LIN {X 0,Y 395.953,Z 958.615,A -85,B 0,C 180,E1 18668.249,E2 18668.249} C_VEL
LIN {X 0,Y 392.265,Z 977.783,A -85,B 0,C 180,E1 18665.892,E2 18665.892} C_VEL
LIN {X 0,Y 388.745,Z 995.88,A -85,B 0,C 180,E1 18663.291,E2 18663.291} C_VEL
LIN {X 0,Y 385.497,Z 1013.366,A -85,B 0,C 180,E1 18660.383,E2 18660.383} C_VEL
LIN {X 0,Y 382.925,Z 1028.309,A -85,B 0,C 180,E1 18657.527,E2 18657.527} C_VEL
LIN {X 0,Y 380.669,Z 1042.529,A -85,B 0,C 180,E1 18654.354,E2 18654.354} C_VEL
LIN {X 0,Y 378.971,Z 1054.652,A -85,B 0,C 180,E1 18651.19,E2 18651.19} C_VEL
LIN {X 0,Y 377.875,Z 1063.785,A -85,B 0,C 180,E1 18648.353,E2 18648.353} C_VEL
LIN {X 0,Y 376.991,Z 1072.565,A -85,B 0,C 180,E1 18645.065,E2 18645.065} C_VEL
LIN {X 0,Y 376.551,Z 1078.821,A -85,B 0,C 180,E1 18642.109,E2 18642.109} C_VEL
LIN {X 0,Y 376.293,Z 1084.179,A -85,B 0,C 180,E1 18638.865,E2 18638.865} C_VEL
LIN {X 0,Y 376.216,Z 1087.581,A -85,B 0,C 180,E1 18635.796,E2 18635.796} C_VEL
LIN {X 0,Y 376.187,Z 1089.458,A -85,B 0,C 180,E1 18633.047,E2 18633.047} C_VEL
LIN {X 0,Y 376.206,Z 1090.251,A -85,B 0,C 180,E1 18630,E2 18630} C_VEL
LIN {X 0,Y 376.187,Z 1089.461,A -85,B 0,C 180,E1 18626.953,E2 18626.953} C_VEL
LIN {X 0,Y 376.215,Z 1087.586,A -85,B 0,C 180,E1 18624.204,E2 18624.204} C_VEL
LIN {X 0,Y 376.297,Z 1083.964,A -85,B 0,C 180,E1 18620.98,E2 18620.98} C_VEL
LIN {X 0,Y 376.573,Z 1078.539,A -85,B 0,C 180,E1 18617.736,E2 18617.736} C_VEL
LIN {X 0,Y 377.088,Z 1071.485,A -85,B 0,C 180,E1 18614.466,E2 18614.466} C_VEL
LIN {X 0,Y 378,Z 1062.621,A -85,B 0,C 180,E1 18611.253,E2 18611.253} C_VEL
LIN {X 0,Y 379.354,Z 1051.878,A -85,B 0,C 180,E1 18608.021,E2 18608.021} C_VEL
LIN {X 0,Y 380.971,Z 1040.525,A -85,B 0,C 180,E1 18605.17,E2 18605.17} C_VEL
LIN {X 0,Y 383.492,Z 1024.877,A -85,B 0,C 180,E1 18601.792,E2 18601.792} C_VEL
LIN {X 0,Y 386.339,Z 1008.954,A -85,B 0,C 180,E1 18598.828,E2 18598.828} C_VEL
LIN {X 0,Y 389.531,Z 991.792,A -85,B 0,C 180,E1 18596.091,E2 18596.091} C_VEL
LIN {X 0,Y 393.28,Z 972.35,A -85,B 0,C 180,E1 18593.412,E2 18593.412} C_VEL
LIN {X 0,Y 397.008,Z 953.443,A -85,B 0,C 180,E1 18591.163,E2 18591.163} C_VEL
LIN {X 0,Y 400.919,Z 932.814,A -85,B 0,C 180,E1 18589.082,E2 18589.082} C_VEL
LIN {X 0,Y 404.892,Z 911.134,A -85,B 0,C 180,E1 18587.226,E2 18587.226} C_VEL
LIN {X 0,Y 408.617,Z 889.656,A -85,B 0,C 180,E1 18585.685,E2 18585.685} C_VEL
LIN {X 0,Y 411.957,Z 868.031,A -85,B 0,C 180,E1 18584.424,E2 18584.424} C_VEL
LIN {X 0,Y 415.071,Z 845.276,A -85,B 0,C 180,E1 18583.348,E2 18583.348} C_VEL
LIN {X 0,Y 417.607,Z 823.088,A -85,B 0,C 180,E1 18582.55,E2 18582.55} C_VEL
LIN {X 0,Y 419.585,Z 798.577,A -85,B 0,C 180,E1 18581.9,E2 18581.9} C_VEL
LIN {X 0,Y 428.412,Z 598.085,A -85,B 0,C 180,E1 18577.889,E2 18577.889} C_VEL
LIN {X 0,Y 432.313,Z 505.731,A -85,B 0,C 180,E1 18576.053,E2 18576.053} C_VEL
LIN {X 0,Y 430.788,Z 488.115,A -85,B 0,C 180,E1 18575.366,E2 18575.366} C_VEL
LIN {X 0,Y 419.802,Z 470.98,A -85,B 0,C 180,E1 18573.134,E2 18573.134} C_VEL
LIN {X 0,Y 416.485,Z 465.848,A -85,B 0,C 180,E1 18572.368,E2 18572.368} C_VEL
LIN {X 0,Y 408.57,Z 450.774,A -85,B 0,C 180,E1 18569.303,E2 18569.303} C_VEL
LIN {X 0,Y 402.669,Z 440.538,A -85,B 0,C 180,E1 18566.866,E2 18566.866} C_VEL
LIN {X 0,Y 398.101,Z 432.532,A -85,B 0,C 180,E1 18564.798,E2 18564.798} C_VEL
LIN {X 0,Y 394.857,Z 427.301,A -85,B 0,C 180,E1 18563.267,E2 18563.267} C_VEL
LIN {X 0,Y 391.803,Z 422.309,A -85,B 0,C 180,E1 18561.717,E2 18561.717} C_VEL
LIN {X 0,Y 389.222,Z 418.314,A -85,B 0,C 180,E1 18560.34,E2 18560.34} C_VEL
LIN {X 0,Y 388.405,Z 416.892,A -85,B 0,C 180,E1 18559.864,E2 18559.864} C_VEL
LIN {X 0,Y 385.879,Z 413.274,A -85,B 0,C 180,E1 18558.428,E2 18558.428} C_VEL
LIN {X 0,Y 385.059,Z 411.546,A -85,B 0,C 180,E1 18557.842,E2 18557.842} C_VEL
LIN {X 0,Y 382.366,Z 408.271,A -85,B 0,C 180,E1 18556.248,E2 18556.248} C_VEL
LIN {X 0,Y 381.062,Z 405.625,A -85,B 0,C 180,E1 18555.211,E2 18555.211} C_VEL
LIN {X 0,Y 378.291,Z 402.297,A -85,B 0,C 180,E1 18553.294,E2 18553.294} C_VEL
LIN {X 0,Y 377.687,Z 400.258,A -85,B 0,C 180,E1 18552.347,E2 18552.347} C_VEL
LIN {X 0,Y 377.63,Z 399.995,A -85,B 0,C 180,E1 18548.987,E2 18548.987} C_VEL
LIN {X 0,Y 377.616,Z 399.995,A -85,B 0,C 180,E1 18545.165,E2 18545.165} C_VEL
LIN {X 0,Y 377.616,Z 399.993,A -85,B 0,C 180,E1 18541.062,E2 18541.062} C_VEL
LIN {X 0,Y 377.616,Z 399.992,A -85,B 0,C 180,E1 18536.964,E2 18536.964} C_VEL
LIN {X 0,Y 377.616,Z 399.989,A -85,B 0,C 180,E1 18532.851,E2 18532.851} C_VEL
LIN {X 0,Y 377.623,Z 399.989,A -85,B 0,C 180,E1 18528.855,E2 18528.855} C_VEL
LIN {X 0,Y 377.637,Z 399.988,A -85,B 0,C 180,E1 18524.961,E2 18524.961} C_VEL
LIN {X 0,Y 377.652,Z 399.988,A -85,B 0,C 180,E1 18520.995,E2 18520.995} C_VEL
LIN {X 0,Y 377.652,Z 400.221,A -85,B 0,C 180,E1 18518.08,E2 18518.08} C_VEL
LIN {X 0,Y 379.501,Z 404.243,A -85,B 0,C 180,E1 18516.062,E2 18516.062} C_VEL
LIN {X 0,Y 381.324,Z 406.087,A -85,B 0,C 180,E1 18514.863,E2 18514.863} C_VEL
LIN {X 0,Y 382.924,Z 409.558,A -85,B 0,C 180,E1 18513.48,E2 18513.48} C_VEL
LIN {X 0,Y 384.703,Z 411.566,A -85,B 0,C 180,E1 18512.409,E2 18512.409} C_VEL
LIN {X 0,Y 386.855,Z 415.598,A -85,B 0,C 180,E1 18510.879,E2 18510.879} C_VEL
LIN {X 0,Y 388.007,Z 417.315,A -85,B 0,C 180,E1 18510.175,E2 18510.175} C_VEL
LIN {X 0,Y 391.15,Z 422.892,A -85,B 0,C 180,E1 18508.225,E2 18508.225} C_VEL
LIN {X 0,Y 393.971,Z 427.927,A -85,B 0,C 180,E1 18506.583,E2 18506.583} C_VEL
LIN {X 0,Y 396.924,Z 433.413,A -85,B 0,C 180,E1 18504.946,E2 18504.946} C_VEL
LIN {X 0,Y 401.486,Z 441.984,A -85,B 0,C 180,E1 18502.579,E2 18502.579} C_VEL
LIN {X 0,Y 407.169,Z 453.602,A -85,B 0,C 180,E1 18499.771,E2 18499.771} C_VEL
LIN {X 0,Y 413.175,Z 466.753,A -85,B 0,C 180,E1 18496.956,E2 18496.956} C_VEL
LIN {X 0,Y 414.811,Z 470.097,A -85,B 0,C 180,E1 18496.371,E2 18496.371} C_VEL
LIN {X 0,Y 422.176,Z 481.769,A -85,B 0,C 180,E1 18494.82,E2 18494.82} C_VEL
LIN {X 0,Y 426.207,Z 512.164,A -85,B 0,C 180,E1 18493.447,E2 18493.447} C_VEL
LIN {X 0,Y 419.079,Z 748.452,A -85,B 0,C 180,E1 18489.374,E2 18489.374} C_VEL
LIN {X 0,Y 417.798,Z 768.888,A -85,B 0,C 180,E1 18488.782,E2 18488.782} C_VEL
LIN {X 0,Y 415.904,Z 788.515,A -85,B 0,C 180,E1 18487.984,E2 18487.984} C_VEL
LIN {X 0,Y 413.573,Z 806.905,A -85,B 0,C 180,E1 18487.013,E2 18487.013} C_VEL
LIN {X 0,Y 410.543,Z 825.493,A -85,B 0,C 180,E1 18485.769,E2 18485.769} C_VEL
LIN {X 0,Y 407.124,Z 843.157,A -85,B 0,C 180,E1 18484.308,E2 18484.308} C_VEL
LIN {X 0,Y 403.192,Z 860.843,A -85,B 0,C 180,E1 18482.525,E2 18482.525} C_VEL
LIN {X 0,Y 399.371,Z 876.448,A -85,B 0,C 180,E1 18480.622,E2 18480.622} C_VEL
LIN {X 0,Y 395.306,Z 891.616,A -85,B 0,C 180,E1 18478.393,E2 18478.393} C_VEL
LIN {X 0,Y 393.493,Z 897.983,A -85,B 0,C 180,E1 18477.31,E2 18477.31} C_VEL
LIN {X 0,Y 391.285,Z 902.98,A -85,B 0,C 180,E1 18476.504,E2 18476.504} C_VEL
LIN {X 0,Y 382.56,Z 915.406,A -85,B 0,C 180,E1 18474.535,E2 18474.535} C_VEL
LIN {X 0,Y 380.407,Z 919.642,A -85,B 0,C 180,E1 18473.623,E2 18473.623} C_VEL
LIN {X 0,Y 377.243,Z 930.013,A -85,B 0,C 180,E1 18470.803,E2 18470.803} C_VEL
LIN {X 0,Y 374.496,Z 939.227,A -85,B 0,C 180,E1 18467.72,E2 18467.72} C_VEL
LIN {X 0,Y 372.489,Z 946.593,A -85,B 0,C 180,E1 18464.615,E2 18464.615} C_VEL
LIN {X 0,Y 370.947,Z 952.787,A -85,B 0,C 180,E1 18461.191,E2 18461.191} C_VEL
LIN {X 0,Y 370.038,Z 957.128,A -85,B 0,C 180,E1 18457.765,E2 18457.765} C_VEL
LIN {X 0,Y 369.539,Z 959.825,A -85,B 0,C 180,E1 18454.345,E2 18454.345} C_VEL
LIN {X 0,Y 369.359,Z 960.993,A -85,B 0,C 180,E1 18450.931,E2 18450.931} C_VEL
LIN {X 0,Y 369.406,Z 960.688,A -85,B 0,C 180,E1 18447.518,E2 18447.518} C_VEL
LIN {X 0,Y 369.689,Z 959.027,A -85,B 0,C 180,E1 18444.257,E2 18444.257} C_VEL
LIN {X 0,Y 370.331,Z 955.662,A -85,B 0,C 180,E1 18440.834,E2 18440.834} C_VEL
LIN {X 0,Y 371.377,Z 950.872,A -85,B 0,C 180,E1 18437.562,E2 18437.562} C_VEL
LIN {X 0,Y 373.071,Z 944.401,A -85,B 0,C 180,E1 18434.295,E2 18434.295} C_VEL
LIN {X 0,Y 375.304,Z 936.512,A -85,B 0,C 180,E1 18431.194,E2 18431.194} C_VEL
LIN {X 0,Y 378.123,Z 927.246,A -85,B 0,C 180,E1 18428.272,E2 18428.272} C_VEL
LIN {X 0,Y 381.56,Z 916,A -85,B 0,C 180,E1 18425.409,E2 18425.409} C_VEL
LIN {X 0,Y 385.313,Z 903.641,A -85,B 0,C 180,E1 18422.825,E2 18422.825} C_VEL
LIN {X 0,Y 389.315,Z 890.006,A -85,B 0,C 180,E1 18420.455,E2 18420.455} C_VEL
LIN {X 0,Y 393.299,Z 875.817,A -85,B 0,C 180,E1 18418.392,E2 18418.392} C_VEL
LIN {X 0,Y 397.328,Z 859.912,A -85,B 0,C 180,E1 18416.471,E2 18416.471} C_VEL
LIN {X 0,Y 401.185,Z 843.001,A -85,B 0,C 180,E1 18414.784,E2 18414.784} C_VEL
LIN {X 0,Y 404.796,Z 824.782,A -85,B 0,C 180,E1 18413.291,E2 18413.291} C_VEL
LIN {X 0,Y 407.854,Z 806.475,A -85,B 0,C 180,E1 18412.073,E2 18412.073} C_VEL
LIN {X 0,Y 410.397,Z 786.949,A -85,B 0,C 180,E1 18411.055,E2 18411.055} C_VEL
LIN {X 0,Y 412.29,Z 767.123,A -85,B 0,C 180,E1 18410.278,E2 18410.278} C_VEL
LIN {X 0,Y 413.536,Z 745.732,A -85,B 0,C 180,E1 18409.69,E2 18409.69} C_VEL
LIN {X 0,Y 420.978,Z 512.412,A -85,B 0,C 180,E1 18405.623,E2 18405.623} C_VEL
LIN {X 0,Y 417.279,Z 485.839,A -85,B 0,C 180,E1 18404.353,E2 18404.353} C_VEL
LIN {X 0,Y 406.186,Z 468.485,A -85,B 0,C 180,E1 18401.843,E2 18401.843} C_VEL
LIN {X 0,Y 399.907,Z 454.656,A -85,B 0,C 180,E1 18398.732,E2 18398.732} C_VEL
LIN {X 0,Y 393.543,Z 441.944,A -85,B 0,C 180,E1 18395.4,E2 18395.4} C_VEL
LIN {X 0,Y 388.521,Z 432.569,A -85,B 0,C 180,E1 18392.539,E2 18392.539} C_VEL
LIN {X 0,Y 385.533,Z 427.329,A -85,B 0,C 180,E1 18390.725,E2 18390.725} C_VEL
LIN {X 0,Y 382.719,Z 422.434,A -85,B 0,C 180,E1 18388.903,E2 18388.903} C_VEL
LIN {X 0,Y 380.492,Z 418.59,A -85,B 0,C 180,E1 18387.351,E2 18387.351} C_VEL
LIN {X 0,Y 379.383,Z 417.056,A -85,B 0,C 180,E1 18386.618,E2 18386.618} C_VEL
LIN {X 0,Y 377.296,Z 413.466,A -85,B 0,C 180,E1 18384.997,E2 18384.997} C_VEL
LIN {X 0,Y 376.589,Z 412.171,A -85,B 0,C 180,E1 18384.4,E2 18384.4} C_VEL
LIN {X 0,Y 374.291,Z 409.186,A -85,B 0,C 180,E1 18382.624,E2 18382.624} C_VEL
LIN {X 0,Y 373.146,Z 406.648,A -85,B 0,C 180,E1 18381.372,E2 18381.372} C_VEL
LIN {X 0,Y 370.453,Z 403.451,A -85,B 0,C 180,E1 18378.898,E2 18378.898} C_VEL
LIN {X 0,Y 369.729,Z 401.266,A -85,B 0,C 180,E1 18377.469,E2 18377.469} C_VEL
LIN {X 0,Y 369.696,Z 400.982,A -85,B 0,C 180,E1 18373.929,E2 18373.929} C_VEL
LIN {X 0,Y 369.707,Z 400.983,A -85,B 0,C 180,E1 18369.968,E2 18369.968} C_VEL
LIN {X 0,Y 369.728,Z 400.983,A -85,B 0,C 180,E1 18366.055,E2 18366.055} C_VEL
LIN {X 0,Y 369.724,Z 400.991,A -85,B 0,C 180,E1 18361.86,E2 18361.86} C_VEL
LIN {X 0,Y 369.726,Z 400.995,A -85,B 0,C 180,E1 18357.831,E2 18357.831} C_VEL
LIN {X 0,Y 369.732,Z 400.985,A -85,B 0,C 180,E1 18353.635,E2 18353.635} C_VEL
LIN {X 0,Y 369.76,Z 401.367,A -85,B 0,C 180,E1 18351.917,E2 18351.917} C_VEL
LIN {X 0,Y 371.469,Z 405.049,A -85,B 0,C 180,E1 18349.611,E2 18349.611} C_VEL
LIN {X 0,Y 373.93,Z 407.588,A -85,B 0,C 180,E1 18347.649,E2 18347.649} C_VEL
LIN {X 0,Y 375.529,Z 410.9,A -85,B 0,C 180,E1 18346.136,E2 18346.136} C_VEL
LIN {X 0,Y 377.622,Z 412.957,A -85,B 0,C 180,E1 18344.804,E2 18344.804} C_VEL
LIN {X 0,Y 379.517,Z 416.766,A -85,B 0,C 180,E1 18343.312,E2 18343.312} C_VEL
LIN {X 0,Y 381.508,Z 419.143,A -85,B 0,C 180,E1 18342.144,E2 18342.144} C_VEL
LIN {X 0,Y 383.837,Z 423.105,A -85,B 0,C 180,E1 18340.682,E2 18340.682} C_VEL
LIN {X 0,Y 384.918,Z 424.474,A -85,B 0,C 180,E1 18340.106,E2 18340.106} C_VEL
LIN {X 0,Y 387.446,Z 428.741,A -85,B 0,C 180,E1 18338.663,E2 18338.663} C_VEL
LIN {X 0,Y 391.868,Z 436.022,A -85,B 0,C 180,E1 18336.386,E2 18336.386} C_VEL
LIN {X 0,Y 396.912,Z 444.518,A -85,B 0,C 180,E1 18334.004,E2 18334.004} C_VEL
LIN {X 0,Y 403.918,Z 457.005,A -85,B 0,C 180,E1 18330.976,E2 18330.976} C_VEL
LIN {X 0,Y 409.473,Z 467.437,A -85,B 0,C 180,E1 18328.825,E2 18328.825} C_VEL
LIN {X 0,Y 420.241,Z 483.599,A -85,B 0,C 180,E1 18326.456,E2 18326.456} C_VEL
LIN {X 0,Y 425.977,Z 493.065,A -85,B 0,C 180,E1 18325.265,E2 18325.265} C_VEL
LIN {X 0,Y 427.038,Z 509.78,A -85,B 0,C 180,E1 18324.654,E2 18324.654} C_VEL
LIN {X 0,Y 418.292,Z 699.403,A -85,B 0,C 180,E1 18320.873,E2 18320.873} C_VEL
LIN {X 0,Y 413.473,Z 803.159,A -85,B 0,C 180,E1 18318.752,E2 18318.752} C_VEL
LIN {X 0,Y 411.266,Z 826.625,A -85,B 0,C 180,E1 18318.074,E2 18318.074} C_VEL
LIN {X 0,Y 408.429,Z 849.45,A -85,B 0,C 180,E1 18317.2,E2 18317.2} C_VEL
LIN {X 0,Y 405.385,Z 870.149,A -85,B 0,C 180,E1 18316.174,E2 18316.174} C_VEL
LIN {X 0,Y 401.415,Z 893.749,A -85,B 0,C 180,E1 18314.722,E2 18314.722} C_VEL
LIN {X 0,Y 397.456,Z 915.589,A -85,B 0,C 180,E1 18313.079,E2 18313.079} C_VEL
LIN {X 0,Y 393.489,Z 935.753,A -85,B 0,C 180,E1 18311.254,E2 18311.254} C_VEL
LIN {X 0,Y 389.176,Z 956.855,A -85,B 0,C 180,E1 18309.01,E2 18309.01} C_VEL
LIN {X 0,Y 385.305,Z 975.879,A -85,B 0,C 180,E1 18306.645,E2 18306.645} C_VEL
LIN {X 0,Y 381.578,Z 993.911,A -85,B 0,C 180,E1 18304.015,E2 18304.015} C_VEL
LIN {X 0,Y 378.118,Z 1011.528,A -85,B 0,C 180,E1 18301.04,E2 18301.04} C_VEL
LIN {X 0,Y 375.369,Z 1026.455,A -85,B 0,C 180,E1 18298.13,E2 18298.13} C_VEL
LIN {X 0,Y 373.078,Z 1039.95,A -85,B 0,C 180,E1 18295.052,E2 18295.052} C_VEL
LIN {X 0,Y 371.263,Z 1052.24,A -85,B 0,C 180,E1 18291.818,E2 18291.818} C_VEL
LIN {X 0,Y 370.023,Z 1062.017,A -85,B 0,C 180,E1 18288.757,E2 18288.757} C_VEL
LIN {X 0,Y 369.137,Z 1070.586,A -85,B 0,C 180,E1 18285.555,E2 18285.555} C_VEL
LIN {X 0,Y 368.654,Z 1077.294,A -85,B 0,C 180,E1 18282.372,E2 18282.372} C_VEL
LIN {X 0,Y 368.381,Z 1082.73,A -85,B 0,C 180,E1 18279.057,E2 18279.057} C_VEL
LIN {X 0,Y 368.325,Z 1086.179,A -85,B 0,C 180,E1 18275.921,E2 18275.921} C_VEL
LIN {X 0,Y 368.3,Z 1088.082,A -85,B 0,C 180,E1 18273.112,E2 18273.112} C_VEL
LIN {X 0,Y 368.323,Z 1088.885,A -85,B 0,C 180,E1 18270,E2 18270} C_VEL
LIN {X 0,Y 368.299,Z 1088.085,A -85,B 0,C 180,E1 18266.887,E2 18266.887} C_VEL
LIN {X 0,Y 368.324,Z 1086.183,A -85,B 0,C 180,E1 18264.079,E2 18264.079} C_VEL
LIN {X 0,Y 368.385,Z 1082.503,A -85,B 0,C 180,E1 18260.785,E2 18260.785} C_VEL
LIN {X 0,Y 368.653,Z 1077.303,A -85,B 0,C 180,E1 18257.628,E2 18257.628} C_VEL
LIN {X 0,Y 369.137,Z 1070.59,A -85,B 0,C 180,E1 18254.445,E2 18254.445} C_VEL
LIN {X 0,Y 370.022,Z 1062.038,A -85,B 0,C 180,E1 18251.243,E2 18251.243} C_VEL
LIN {X 0,Y 371.343,Z 1051.707,A -85,B 0,C 180,E1 18248.021,E2 18248.021} C_VEL
LIN {X 0,Y 373.188,Z 1039.297,A -85,B 0,C 180,E1 18244.786,E2 18244.786} C_VEL
LIN {X 0,Y 375.643,Z 1024.859,A -85,B 0,C 180,E1 18241.546,E2 18241.546} C_VEL
LIN {X 0,Y 378.467,Z 1009.78,A -85,B 0,C 180,E1 18238.637,E2 18238.637} C_VEL
LIN {X 0,Y 381.743,Z 993.089,A -85,B 0,C 180,E1 18235.859,E2 18235.859} C_VEL
LIN {X 0,Y 385.401,Z 975.349,A -85,B 0,C 180,E1 18233.287,E2 18233.287} C_VEL
LIN {X 0,Y 389.317,Z 956.164,A -85,B 0,C 180,E1 18230.912,E2 18230.912} C_VEL
LIN {X 0,Y 393.637,Z 934.916,A -85,B 0,C 180,E1 18228.668,E2 18228.668} C_VEL
LIN {X 0,Y 397.708,Z 914.187,A -85,B 0,C 180,E1 18226.808,E2 18226.808} C_VEL
LIN {X 0,Y 401.607,Z 892.632,A -85,B 0,C 180,E1 18225.205,E2 18225.205} C_VEL
LIN {X 0,Y 405.493,Z 869.313,A -85,B 0,C 180,E1 18223.785,E2 18223.785} C_VEL
LIN {X 0,Y 408.67,Z 847.644,A -85,B 0,C 180,E1 18222.721,E2 18222.721} C_VEL
LIN {X 0,Y 411.442,Z 824.725,A -85,B 0,C 180,E1 18221.866,E2 18221.866} C_VEL
LIN {X 0,Y 413.62,Z 800.142,A -85,B 0,C 180,E1 18221.185,E2 18221.185} C_VEL
LIN {X 0,Y 422.674,Z 603.781,A -85,B 0,C 180,E1 18217.214,E2 18217.214} C_VEL
LIN {X 0,Y 426.949,Z 507.051,A -85,B 0,C 180,E1 18215.274,E2 18215.274} C_VEL
LIN {X 0,Y 425.762,Z 492.469,A -85,B 0,C 180,E1 18214.7,E2 18214.7} C_VEL
LIN {X 0,Y 415.332,Z 476.131,A -85,B 0,C 180,E1 18212.509,E2 18212.509} C_VEL
LIN {X 0,Y 408.557,Z 465.902,A -85,B 0,C 180,E1 18210.925,E2 18210.925} C_VEL
LIN {X 0,Y 401.234,Z 452.26,A -85,B 0,C 180,E1 18207.936,E2 18207.936} C_VEL
LIN {X 0,Y 395.316,Z 441.89,A -85,B 0,C 180,E1 18205.305,E2 18205.305} C_VEL
LIN {X 0,Y 390.672,Z 433.961,A -85,B 0,C 180,E1 18203.052,E2 18203.052} C_VEL
LIN {X 0,Y 387.343,Z 428.643,A -85,B 0,C 180,E1 18201.343,E2 18201.343} C_VEL
LIN {X 0,Y 384.807,Z 424.315,A -85,B 0,C 180,E1 18199.9,E2 18199.9} C_VEL
LIN {X 0,Y 381.799,Z 419.925,A -85,B 0,C 180,E1 18198.157,E2 18198.157} C_VEL
LIN {X 0,Y 380.943,Z 418.281,A -85,B 0,C 180,E1 18197.568,E2 18197.568} C_VEL
LIN {X 0,Y 378.156,Z 414.514,A -85,B 0,C 180,E1 18195.803,E2 18195.803} C_VEL
LIN {X 0,Y 377.263,Z 412.608,A -85,B 0,C 180,E1 18195.053,E2 18195.053} C_VEL
LIN {X 0,Y 374.512,Z 409.275,A -85,B 0,C 180,E1 18193.116,E2 18193.116} C_VEL
LIN {X 0,Y 373.492,Z 406.896,A -85,B 0,C 180,E1 18192.052,E2 18192.052} C_VEL
LIN {X 0,Y 370.312,Z 403.262,A -85,B 0,C 180,E1 18189.323,E2 18189.323} C_VEL
LIN {X 0,Y 369.737,Z 401.228,A -85,B 0,C 180,E1 18188.083,E2 18188.083} C_VEL
LIN {X 0,Y 369.716,Z 400.97,A -85,B 0,C 180,E1 18184.342,E2 18184.342} C_VEL
LIN {X 0,Y 369.729,Z 400.97,A -85,B 0,C 180,E1 18180.154,E2 18180.154} C_VEL
LIN {X 0,Y 369.719,Z 400.974,A -85,B 0,C 180,E1 18175.968,E2 18175.968} C_VEL
LIN {X 0,Y 369.719,Z 400.976,A -85,B 0,C 180,E1 18171.915,E2 18171.915} C_VEL
LIN {X 0,Y 369.711,Z 400.981,A -85,B 0,C 180,E1 18167.822,E2 18167.822} C_VEL
LIN {X 0,Y 369.691,Z 400.985,A -85,B 0,C 180,E1 18163.986,E2 18163.986} C_VEL
LIN {X 0,Y 369.746,Z 401.397,A -85,B 0,C 180,E1 18162.153,E2 18162.153} C_VEL
LIN {X 0,Y 371.75,Z 405.408,A -85,B 0,C 180,E1 18159.534,E2 18159.534} C_VEL
LIN {X 0,Y 373.611,Z 407.403,A -85,B 0,C 180,E1 18157.996,E2 18157.996} C_VEL
LIN {X 0,Y 375.537,Z 411.187,A -85,B 0,C 180,E1 18156.127,E2 18156.127} C_VEL
LIN {X 0,Y 377.096,Z 412.832,A -85,B 0,C 180,E1 18155.065,E2 18155.065} C_VEL
LIN {X 0,Y 378.908,Z 416.518,A -85,B 0,C 180,E1 18153.515,E2 18153.515} C_VEL
LIN {X 0,Y 380.346,Z 418.233,A -85,B 0,C 180,E1 18152.61,E2 18152.61} C_VEL
LIN {X 0,Y 382.737,Z 422.484,A -85,B 0,C 180,E1 18150.928,E2 18150.928} C_VEL
LIN {X 0,Y 386.507,Z 429.147,A -85,B 0,C 180,E1 18148.496,E2 18148.496} C_VEL
LIN {X 0,Y 389.531,Z 434.715,A -85,B 0,C 180,E1 18146.681,E2 18146.681} C_VEL
LIN {X 0,Y 392.449,Z 440.19,A -85,B 0,C 180,E1 18145.023,E2 18145.023} C_VEL
LIN {X 0,Y 397.596,Z 449.955,A -85,B 0,C 180,E1 18142.331,E2 18142.331} C_VEL
LIN {X 0,Y 403.825,Z 463.23,A -85,B 0,C 180,E1 18139.182,E2 18139.182} C_VEL
LIN {X 0,Y 406.872,Z 469.685,A -85,B 0,C 180,E1 18137.841,E2 18137.841} C_VEL
LIN {X 0,Y 417.414,Z 486.175,A -85,B 0,C 180,E1 18135.509,E2 18135.509} C_VEL
LIN {X 0,Y 420.937,Z 513.738,A -85,B 0,C 180,E1 18134.244,E2 18134.244} C_VEL
LIN {X 0,Y 413.382,Z 749.141,A -85,B 0,C 180,E1 18130.141,E2 18130.141} C_VEL
LIN {X 0,Y 412.046,Z 769.564,A -85,B 0,C 180,E1 18129.544,E2 18129.544} C_VEL
LIN {X 0,Y 409.972,Z 790.073,A -85,B 0,C 180,E1 18128.699,E2 18128.699} C_VEL
LIN {X 0,Y 407.408,Z 809.098,A -85,B 0,C 180,E1 18127.669,E2 18127.669} C_VEL
LIN {X 0,Y 404.271,Z 827.544,A -85,B 0,C 180,E1 18126.412,E2 18126.412} C_VEL
LIN {X 0,Y 400.714,Z 845.004,A -85,B 0,C 180,E1 18124.935,E2 18124.935} C_VEL
LIN {X 0,Y 396.683,Z 862.318,A -85,B 0,C 180,E1 18123.159,E2 18123.159} C_VEL
LIN {X 0,Y 392.644,Z 878.07,A -85,B 0,C 180,E1 18121.204,E2 18121.204} C_VEL
LIN {X 0,Y 388.412,Z 893.187,A -85,B 0,C 180,E1 18118.944,E2 18118.944} C_VEL
LIN {X 0,Y 384.46,Z 906.431,A -85,B 0,C 180,E1 18116.538,E2 18116.538} C_VEL
LIN {X 0,Y 380.884,Z 918.065,A -85,B 0,C 180,E1 18114.001,E2 18114.001} C_VEL
LIN {X 0,Y 380.407,Z 919.642,A -85,B 0,C 180,E1 18113.623,E2 18113.623} C_VEL
LIN {X 0,Y 378.303,Z 923.784,A -85,B 0,C 180,E1 18112.683,E2 18112.683} C_VEL
LIN {X 0,Y 369.926,Z 934,A -85,B 0,C 180,E1 18110.348,E2 18110.348} C_VEL
LIN {X 0,Y 367.984,Z 937.352,A -85,B 0,C 180,E1 18109.309,E2 18109.309} C_VEL
LIN {X 0,Y 365.499,Z 945.595,A -85,B 0,C 180,E1 18106.039,E2 18106.039} C_VEL
LIN {X 0,Y 363.606,Z 952.398,A -85,B 0,C 180,E1 18102.525,E2 18102.525} C_VEL
LIN {X 0,Y 362.499,Z 957.108,A -85,B 0,C 180,E1 18099.206,E2 18099.206} C_VEL
LIN {X 0,Y 361.824,Z 960.439,A -85,B 0,C 180,E1 18095.709,E2 18095.709} C_VEL
LIN {X 0,Y 361.523,Z 962.134,A -85,B 0,C 180,E1 18092.219,E2 18092.219} C_VEL
LIN {X 0,Y 361.477,Z 962.352,A -85,B 0,C 180,E1 18088.891,E2 18088.891} C_VEL
LIN {X 0,Y 361.694,Z 961.065,A -85,B 0,C 180,E1 18085.243,E2 18085.243} C_VEL
LIN {X 0,Y 362.253,Z 958.266,A -85,B 0,C 180,E1 18081.748,E2 18081.748} C_VEL
LIN {X 0,Y 363.214,Z 954.087,A -85,B 0,C 180,E1 18078.407,E2 18078.407} C_VEL
LIN {X 0,Y 364.882,Z 947.877,A -85,B 0,C 180,E1 18074.911,E2 18074.911} C_VEL
LIN {X 0,Y 367.021,Z 940.486,A -85,B 0,C 180,E1 18071.742,E2 18071.742} C_VEL
LIN {X 0,Y 369.939,Z 931.251,A -85,B 0,C 180,E1 18068.6,E2 18068.6} C_VEL
LIN {X 0,Y 373.392,Z 920.516,A -85,B 0,C 180,E1 18065.646,E2 18065.646} C_VEL
LIN {X 0,Y 377.135,Z 909.019,A -85,B 0,C 180,E1 18063.041,E2 18063.041} C_VEL
LIN {X 0,Y 381.34,Z 895.476,A -85,B 0,C 180,E1 18060.516,E2 18060.516} C_VEL
LIN {X 0,Y 385.677,Z 880.742,A -85,B 0,C 180,E1 18058.246,E2 18058.246} C_VEL
LIN {X 0,Y 390.017,Z 864.744,A -85,B 0,C 180,E1 18056.199,E2 18056.199} C_VEL
LIN {X 0,Y 394.032,Z 848.495,A -85,B 0,C 180,E1 18054.472,E2 18054.472} C_VEL
LIN {X 0,Y 397.883,Z 830.546,A -85,B 0,C 180,E1 18052.907,E2 18052.907} C_VEL
LIN {X 0,Y 401.132,Z 812.506,A -85,B 0,C 180,E1 18051.636,E2 18051.636} C_VEL
LIN {X 0,Y 404.051,Z 792.438,A -85,B 0,C 180,E1 18050.508,E2 18050.508} C_VEL
LIN {X 0,Y 406.211,Z 772.796,A -85,B 0,C 180,E1 18049.663,E2 18049.663} C_VEL
LIN {X 0,Y 407.695,Z 751.968,A -85,B 0,C 180,E1 18049.025,E2 18049.025} C_VEL
LIN {X 0,Y 408.852,Z 717.479,A -85,B 0,C 180,E1 18048.373,E2 18048.373} C_VEL
LIN {X 0,Y 415.809,Z 514.095,A -85,B 0,C 180,E1 18044.81,E2 18044.81} C_VEL
LIN {X 0,Y 412.604,Z 490.462,A -85,B 0,C 180,E1 18043.657,E2 18043.657} C_VEL
LIN {X 0,Y 402.05,Z 473.99,A -85,B 0,C 180,E1 18041.226,E2 18041.226} C_VEL
LIN {X 0,Y 398.237,Z 467.919,A -85,B 0,C 180,E1 18040.185,E2 18040.185} C_VEL
LIN {X 0,Y 392.243,Z 455.192,A -85,B 0,C 180,E1 18037.073,E2 18037.073} C_VEL
LIN {X 0,Y 386.427,Z 443.595,A -85,B 0,C 180,E1 18033.801,E2 18033.801} C_VEL
LIN {X 0,Y 382.796,Z 437.208,A -85,B 0,C 180,E1 18031.669,E2 18031.669} C_VEL
LIN {X 0,Y 380.93,Z 433.629,A -85,B 0,C 180,E1 18030.437,E2 18030.437} C_VEL
LIN {X 0,Y 378.176,Z 428.788,A -85,B 0,C 180,E1 18028.591,E2 18028.591} C_VEL
LIN {X 0,Y 375.642,Z 424.258,A -85,B 0,C 180,E1 18026.733,E2 18026.733} C_VEL
LIN {X 0,Y 373.341,Z 420.816,A -85,B 0,C 180,E1 18025.034,E2 18025.034} C_VEL
LIN {X 0,Y 372.501,Z 419.004,A -85,B 0,C 180,E1 18024.248,E2 18024.248} C_VEL
LIN {X 0,Y 370.046,Z 415.563,A -85,B 0,C 180,E1 18022.228,E2 18022.228} C_VEL
LIN {X 0,Y 369.035,Z 413.435,A -85,B 0,C 180,E1 18021.122,E2 18021.122} C_VEL
LIN {X 0,Y 366.572,Z 410.423,A -85,B 0,C 180,E1 18018.776,E2 18018.776} C_VEL
LIN {X 0,Y 365.383,Z 407.76,A -85,B 0,C 180,E1 18017.026,E2 18017.026} C_VEL
LIN {X 0,Y 361.832,Z 402.283,A -85,B 0,C 180,E1 18010.343,E2 18010.343} C_VEL
LIN {X 0,Y 361.782,Z 401.967,A -85,B 0,C 180,E1 18006.347,E2 18006.347} C_VEL
LIN {X 0,Y 361.777,Z 401.979,A -85,B 0,C 180,E1 18002.218,E2 18002.218} C_VEL
LIN {X 0,Y 361.805,Z 402.374,A -85,B 0,C 180,E1 17999.05,E2 17999.05} C_VEL
LIN {X 0,Y 366.116,Z 408.659,A -85,B 0,C 180,E1 17991.836,E2 17991.836} C_VEL
LIN {X 0,Y 367.722,Z 412.012,A -85,B 0,C 180,E1 17989.821,E2 17989.821} C_VEL
LIN {X 0,Y 370.153,Z 414.61,A -85,B 0,C 180,E1 17987.838,E2 17987.838} C_VEL
LIN {X 0,Y 371.967,Z 418.116,A -85,B 0,C 180,E1 17986.159,E2 17986.159} C_VEL
LIN {X 0,Y 373.774,Z 420.08,A -85,B 0,C 180,E1 17984.949,E2 17984.949} C_VEL
LIN {X 0,Y 376.195,Z 424.334,A -85,B 0,C 180,E1 17983.16,E2 17983.16} C_VEL
LIN {X 0,Y 377.442,Z 425.802,A -85,B 0,C 180,E1 17982.423,E2 17982.423} C_VEL
LIN {X 0,Y 379.989,Z 430.082,A -85,B 0,C 180,E1 17980.798,E2 17980.798} C_VEL
LIN {X 0,Y 381.44,Z 432.601,A -85,B 0,C 180,E1 17979.917,E2 17979.917} C_VEL
LIN {X 0,Y 384.331,Z 437.192,A -85,B 0,C 180,E1 17978.321,E2 17978.321} C_VEL
LIN {X 0,Y 388.188,Z 443.685,A -85,B 0,C 180,E1 17976.309,E2 17976.309} C_VEL
LIN {X 0,Y 392.581,Z 451.273,A -85,B 0,C 180,E1 17974.182,E2 17974.182} C_VEL
LIN {X 0,Y 399.331,Z 463.429,A -85,B 0,C 180,E1 17971.205,E2 17971.205} C_VEL
LIN {X 0,Y 401.873,Z 467.896,A -85,B 0,C 180,E1 17970.282,E2 17970.282} C_VEL
LIN {X 0,Y 413.499,Z 485.046,A -85,B 0,C 180,E1 17967.575,E2 17967.575} C_VEL
LIN {X 0,Y 420.953,Z 497.215,A -85,B 0,C 180,E1 17965.963,E2 17965.963} C_VEL
LIN {X 0,Y 421.75,Z 511.275,A -85,B 0,C 180,E1 17965.448,E2 17965.448} C_VEL
LIN {X 0,Y 412.649,Z 700.595,A -85,B 0,C 180,E1 17961.643,E2 17961.643} C_VEL
LIN {X 0,Y 407.718,Z 802.375,A -85,B 0,C 180,E1 17959.542,E2 17959.542} C_VEL
LIN {X 0,Y 405.432,Z 825.829,A -85,B 0,C 180,E1 17958.861,E2 17958.861} C_VEL
LIN {X 0,Y 402.454,Z 848.822,A -85,B 0,C 180,E1 17957.974,E2 17957.974} C_VEL
LIN {X 0,Y 399.307,Z 869.335,A -85,B 0,C 180,E1 17956.949,E2 17956.949} C_VEL
LIN {X 0,Y 395.244,Z 892.519,A -85,B 0,C 180,E1 17955.511,E2 17955.511} C_VEL
LIN {X 0,Y 391.243,Z 913.557,A -85,B 0,C 180,E1 17953.925,E2 17953.925} C_VEL
LIN {X 0,Y 386.903,Z 934.504,A -85,B 0,C 180,E1 17952.015,E2 17952.015} C_VEL
LIN {X 0,Y 382.446,Z 955.347,A -85,B 0,C 180,E1 17949.77,E2 17949.77} C_VEL
LIN {X 0,Y 378.272,Z 974.586,A -85,B 0,C 180,E1 17947.346,E2 17947.346} C_VEL
LIN {X 0,Y 374.318,Z 992.776,A -85,B 0,C 180,E1 17944.644,E2 17944.644} C_VEL
LIN {X 0,Y 370.6,Z 1010.625,A -85,B 0,C 180,E1 17941.561,E2 17941.561} C_VEL
LIN {X 0,Y 367.67,Z 1025.666,A -85,B 0,C 180,E1 17938.554,E2 17938.554} C_VEL
LIN {X 0,Y 365.273,Z 1039.06,A -85,B 0,C 180,E1 17935.405,E2 17935.405} C_VEL
LIN {X 0,Y 363.321,Z 1051.635,A -85,B 0,C 180,E1 17931.965,E2 17931.965} C_VEL
LIN {X 0,Y 362.068,Z 1061.229,A -85,B 0,C 180,E1 17928.851,E2 17928.851} C_VEL
LIN {X 0,Y 361.156,Z 1070.032,A -85,B 0,C 180,E1 17925.413,E2 17925.413} C_VEL
LIN {X 0,Y 360.732,Z 1076.043,A -85,B 0,C 180,E1 17922.486,E2 17922.486} C_VEL
LIN {X 0,Y 360.47,Z 1081.482,A -85,B 0,C 180,E1 17919.087,E2 17919.087} C_VEL
LIN {X 0,Y 360.429,Z 1084.908,A -85,B 0,C 180,E1 17915.891,E2 17915.891} C_VEL
LIN {X 0,Y 360.413,Z 1086.783,A -85,B 0,C 180,E1 17913.021,E2 17913.021} C_VEL
LIN {X 0,Y 360.432,Z 1087.502,A -85,B 0,C 180,E1 17909.841,E2 17909.841} C_VEL
LIN {X 0,Y 360.414,Z 1086.707,A -85,B 0,C 180,E1 17906.819,E2 17906.819} C_VEL
LIN {X 0,Y 360.434,Z 1084.781,A -85,B 0,C 180,E1 17903.949,E2 17903.949} C_VEL
LIN {X 0,Y 360.471,Z 1081.027,A -85,B 0,C 180,E1 17900.581,E2 17900.581} C_VEL
LIN {X 0,Y 360.748,Z 1075.695,A -85,B 0,C 180,E1 17897.317,E2 17897.317} C_VEL
LIN {X 0,Y 361.296,Z 1068.567,A -85,B 0,C 180,E1 17893.934,E2 17893.934} C_VEL
LIN {X 0,Y 362.227,Z 1059.804,A -85,B 0,C 180,E1 17890.656,E2 17890.656} C_VEL
LIN {X 0,Y 363.724,Z 1048.791,A -85,B 0,C 180,E1 17887.194,E2 17887.194} C_VEL
LIN {X 0,Y 365.637,Z 1036.903,A -85,B 0,C 180,E1 17884.053,E2 17884.053} C_VEL
LIN {X 0,Y 368.29,Z 1022.293,A -85,B 0,C 180,E1 17880.746,E2 17880.746} C_VEL
LIN {X 0,Y 371.423,Z 1006.688,A -85,B 0,C 180,E1 17877.701,E2 17877.701} C_VEL
LIN {X 0,Y 375.03,Z 989.472,A -85,B 0,C 180,E1 17874.839,E2 17874.839} C_VEL
LIN {X 0,Y 379.177,Z 970.283,A -85,B 0,C 180,E1 17872.091,E2 17872.091} C_VEL
LIN {X 0,Y 383.442,Z 950.86,A -85,B 0,C 180,E1 17869.708,E2 17869.708} C_VEL
LIN {X 0,Y 387.727,Z 930.481,A -85,B 0,C 180,E1 17867.596,E2 17867.596} C_VEL
LIN {X 0,Y 392.179,Z 908.609,A -85,B 0,C 180,E1 17865.688,E2 17865.688} C_VEL
LIN {X 0,Y 396.265,Z 887.128,A -85,B 0,C 180,E1 17864.122,E2 17864.122} C_VEL
LIN {X 0,Y 400.004,Z 864.773,A -85,B 0,C 180,E1 17862.807,E2 17862.807} C_VEL
LIN {X 0,Y 403.563,Z 840.294,A -85,B 0,C 180,E1 17861.669,E2 17861.669} C_VEL
LIN {X 0,Y 406.406,Z 816.994,A -85,B 0,C 180,E1 17860.858,E2 17860.858} C_VEL
LIN {X 0,Y 408.238,Z 793.24,A -85,B 0,C 180,E1 17860.256,E2 17860.256} C_VEL
LIN {X 0,Y 417.891,Z 590.632,A -85,B 0,C 180,E1 17856.138,E2 17856.138} C_VEL
LIN {X 0,Y 421.678,Z 508.474,A -85,B 0,C 180,E1 17854.479,E2 17854.479} C_VEL
LIN {X 0,Y 420.691,Z 496.639,A -85,B 0,C 180,E1 17853.994,E2 17853.994} C_VEL
LIN {X 0,Y 409.358,Z 478.789,A -85,B 0,C 180,E1 17851.513,E2 17851.513} C_VEL
LIN {X 0,Y 400.772,Z 466.323,A -85,B 0,C 180,E1 17849.437,E2 17849.437} C_VEL
LIN {X 0,Y 394.717,Z 454.916,A -85,B 0,C 180,E1 17846.8,E2 17846.8} C_VEL
LIN {X 0,Y 388.396,Z 444.061,A -85,B 0,C 180,E1 17843.839,E2 17843.839} C_VEL
LIN {X 0,Y 385.866,Z 439.827,A -85,B 0,C 180,E1 17842.55,E2 17842.55} C_VEL
LIN {X 0,Y 383.198,Z 435.305,A -85,B 0,C 180,E1 17841.104,E2 17841.104} C_VEL
LIN {X 0,Y 380.146,Z 430.275,A -85,B 0,C 180,E1 17839.354,E2 17839.354} C_VEL
LIN {X 0,Y 377.527,Z 426.105,A -85,B 0,C 180,E1 17837.732,E2 17837.732} C_VEL
LIN {X 0,Y 376.302,Z 424.484,A -85,B 0,C 180,E1 17836.994,E2 17836.994} C_VEL
LIN {X 0,Y 373.827,Z 420.293,A -85,B 0,C 180,E1 17835.195,E2 17835.195} C_VEL
LIN {X 0,Y 370.424,Z 415.547,A -85,B 0,C 180,E1 17832.628,E2 17832.628} C_VEL
LIN {X 0,Y 369.705,Z 413.881,A -85,B 0,C 180,E1 17831.861,E2 17831.861} C_VEL
LIN {X 0,Y 366.597,Z 410.203,A -85,B 0,C 180,E1 17829.101,E2 17829.101} C_VEL
LIN {X 0,Y 365.741,Z 408.066,A -85,B 0,C 180,E1 17827.856,E2 17827.856} C_VEL
LIN {X 0,Y 362.088,Z 403.469,A -85,B 0,C 180,E1 17822.69,E2 17822.69} C_VEL
LIN {X 0,Y 361.772,Z 402.121,A -85,B 0,C 180,E1 17820.633,E2 17820.633} C_VEL
LIN {X 0,Y 361.749,Z 401.965,A -85,B 0,C 180,E1 17816.513,E2 17816.513} C_VEL
LIN {X 0,Y 361.74,Z 401.965,A -85,B 0,C 180,E1 17812.535,E2 17812.535} C_VEL
LIN {X 0,Y 361.814,Z 402.379,A -85,B 0,C 180,E1 17809.007,E2 17809.007} C_VEL
LIN {X 0,Y 365.82,Z 408.436,A -85,B 0,C 180,E1 17802.174,E2 17802.174} C_VEL
LIN {X 0,Y 367.848,Z 412.36,A -85,B 0,C 180,E1 17799.639,E2 17799.639} C_VEL
LIN {X 0,Y 369.516,Z 414.101,A -85,B 0,C 180,E1 17798.241,E2 17798.241} C_VEL
LIN {X 0,Y 371.567,Z 418.127,A -85,B 0,C 180,E1 17796.194,E2 17796.194} C_VEL
LIN {X 0,Y 372.871,Z 419.563,A -85,B 0,C 180,E1 17795.271,E2 17795.271} C_VEL
LIN {X 0,Y 374.917,Z 423.483,A -85,B 0,C 180,E1 17793.553,E2 17793.553} C_VEL
LIN {X 0,Y 376.058,Z 424.988,A -85,B 0,C 180,E1 17792.786,E2 17792.786} C_VEL
LIN {X 0,Y 378.699,Z 429.449,A -85,B 0,C 180,E1 17790.934,E2 17790.934} C_VEL
LIN {X 0,Y 382.117,Z 435.923,A -85,B 0,C 180,E1 17788.62,E2 17788.62} C_VEL
LIN {X 0,Y 384.86,Z 440.979,A -85,B 0,C 180,E1 17786.935,E2 17786.935} C_VEL
LIN {X 0,Y 389.136,Z 449.011,A -85,B 0,C 180,E1 17784.5,E2 17784.5} C_VEL
LIN {X 0,Y 394.8,Z 460.48,A -85,B 0,C 180,E1 17781.463,E2 17781.463} C_VEL
LIN {X 0,Y 399.034,Z 469.548,A -85,B 0,C 180,E1 17779.397,E2 17779.397} C_VEL
LIN {X 0,Y 409.66,Z 485.713,A -85,B 0,C 180,E1 17776.89,E2 17776.89} C_VEL
LIN {X 0,Y 412.781,Z 491.127,A -85,B 0,C 180,E1 17776.187,E2 17776.187} C_VEL
LIN {X 0,Y 415.749,Z 515.367,A -85,B 0,C 180,E1 17775.06,E2 17775.06} C_VEL
LIN {X 0,Y 407.758,Z 749.817,A -85,B 0,C 180,E1 17770.93,E2 17770.93} C_VEL
LIN {X 0,Y 406.369,Z 770.189,A -85,B 0,C 180,E1 17770.33,E2 17770.33} C_VEL
LIN {X 0,Y 404.202,Z 790.812,A -85,B 0,C 180,E1 17769.475,E2 17769.475} C_VEL
LIN {X 0,Y 401.482,Z 810.178,A -85,B 0,C 180,E1 17768.416,E2 17768.416} C_VEL
LIN {X 0,Y 398.224,Z 828.614,A -85,B 0,C 180,E1 17767.146,E2 17767.146} C_VEL
LIN {X 0,Y 394.522,Z 846.066,A -85,B 0,C 180,E1 17765.655,E2 17765.655} C_VEL
LIN {X 0,Y 390.325,Z 863.388,A -85,B 0,C 180,E1 17763.859,E2 17763.859} C_VEL
LIN {X 0,Y 386.128,Z 879.105,A -85,B 0,C 180,E1 17761.887,E2 17761.887} C_VEL
LIN {X 0,Y 381.819,Z 893.838,A -85,B 0,C 180,E1 17759.665,E2 17759.665} C_VEL
LIN {X 0,Y 377.711,Z 907.016,A -85,B 0,C 180,E1 17757.256,E2 17757.256} C_VEL
LIN {X 0,Y 373.775,Z 919.259,A -85,B 0,C 180,E1 17754.561,E2 17754.561} C_VEL
LIN {X 0,Y 370.353,Z 929.922,A -85,B 0,C 180,E1 17751.707,E2 17751.707} C_VEL
LIN {X 0,Y 367.984,Z 937.352,A -85,B 0,C 180,E1 17749.309,E2 17749.309} C_VEL
LIN {X 0,Y 366.109,Z 940.603,A -85,B 0,C 180,E1 17748.247,E2 17748.247} C_VEL
LIN {X 0,Y 358.001,Z 948.89,A -85,B 0,C 180,E1 17745.424,E2 17745.424} C_VEL
LIN {X 0,Y 356.694,Z 950.953,A -85,B 0,C 180,E1 17744.433,E2 17744.433} C_VEL
LIN {X 0,Y 355.121,Z 956.646,A -85,B 0,C 180,E1 17740.874,E2 17740.874} C_VEL
LIN {X 0,Y 354.218,Z 960.613,A -85,B 0,C 180,E1 17737.298,E2 17737.298} C_VEL
LIN {X 0,Y 353.731,Z 962.994,A -85,B 0,C 180,E1 17733.728,E2 17733.728} C_VEL
LIN {X 0,Y 353.591,Z 963.821,A -85,B 0,C 180,E1 17730.162,E2 17730.162} C_VEL
LIN {X 0,Y 353.681,Z 963.196,A -85,B 0,C 180,E1 17726.759,E2 17726.759} C_VEL
LIN {X 0,Y 354.109,Z 961.1,A -85,B 0,C 180,E1 17723.189,E2 17723.189} C_VEL
LIN {X 0,Y 354.907,Z 957.645,A -85,B 0,C 180,E1 17719.777,E2 17719.777} C_VEL
LIN {X 0,Y 356.332,Z 952.34,A -85,B 0,C 180,E1 17716.201,E2 17716.201} C_VEL
LIN {X 0,Y 358.391,Z 945.447,A -85,B 0,C 180,E1 17712.799,E2 17712.799} C_VEL
LIN {X 0,Y 361.103,Z 937.081,A -85,B 0,C 180,E1 17709.581,E2 17709.581} C_VEL
LIN {X 0,Y 364.391,Z 927.309,A -85,B 0,C 180,E1 17706.555,E2 17706.555} C_VEL
LIN {X 0,Y 368.215,Z 916.144,A -85,B 0,C 180,E1 17703.729,E2 17703.729} C_VEL
LIN {X 0,Y 372.489,Z 903.313,A -85,B 0,C 180,E1 17701.054,E2 17701.054} C_VEL
LIN {X 0,Y 376.924,Z 889.338,A -85,B 0,C 180,E1 17698.668,E2 17698.668} C_VEL
LIN {X 0,Y 381.228,Z 874.721,A -85,B 0,C 180,E1 17696.58,E2 17696.58} C_VEL
LIN {X 0,Y 385.606,Z 858.703,A -85,B 0,C 180,E1 17694.674,E2 17694.674} C_VEL
LIN {X 0,Y 389.693,Z 841.805,A -85,B 0,C 180,E1 17693.01,E2 17693.01} C_VEL
LIN {X 0,Y 393.373,Z 823.975,A -85,B 0,C 180,E1 17691.577,E2 17691.577} C_VEL
LIN {X 0,Y 396.775,Z 804.183,A -85,B 0,C 180,E1 17690.296,E2 17690.296} C_VEL
LIN {X 0,Y 399.454,Z 784.454,A -85,B 0,C 180,E1 17689.303,E2 17689.303} C_VEL
LIN {X 0,Y 401.38,Z 764.599,A -85,B 0,C 180,E1 17688.556,E2 17688.556} C_VEL
LIN {X 0,Y 402.505,Z 744.214,A -85,B 0,C 180,E1 17688.028,E2 17688.028} C_VEL
LIN {X 0,Y 410.711,Z 515.652,A -85,B 0,C 180,E1 17683.97,E2 17683.97} C_VEL
LIN {X 0,Y 407.992,Z 495.072,A -85,B 0,C 180,E1 17682.945,E2 17682.945} C_VEL
LIN {X 0,Y 397.704,Z 478.892,A -85,B 0,C 180,E1 17680.486,E2 17680.486} C_VEL
LIN {X 0,Y 390.752,Z 468.476,A -85,B 0,C 180,E1 17678.635,E2 17678.635} C_VEL
LIN {X 0,Y 385.382,Z 457.286,A -85,B 0,C 180,E1 17675.701,E2 17675.701} C_VEL
LIN {X 0,Y 380.932,Z 448.57,A -85,B 0,C 180,E1 17673.09,E2 17673.09} C_VEL
LIN {X 0,Y 378.433,Z 443.912,A -85,B 0,C 180,E1 17671.543,E2 17671.543} C_VEL
LIN {X 0,Y 376.086,Z 439.542,A -85,B 0,C 180,E1 17669.988,E2 17669.988} C_VEL
LIN {X 0,Y 373.762,Z 435.283,A -85,B 0,C 180,E1 17668.343,E2 17668.343} C_VEL
LIN {X 0,Y 371.157,Z 430.696,A -85,B 0,C 180,E1 17666.391,E2 17666.391} C_VEL
LIN {X 0,Y 369.006,Z 427.119,A -85,B 0,C 180,E1 17664.663,E2 17664.663} C_VEL
LIN {X 0,Y 368.318,Z 425.748,A -85,B 0,C 180,E1 17664.029,E2 17664.029} C_VEL
LIN {X 0,Y 365.968,Z 422.261,A -85,B 0,C 180,E1 17661.981,E2 17661.981} C_VEL
LIN {X 0,Y 365.007,Z 420.281,A -85,B 0,C 180,E1 17660.916,E2 17660.916} C_VEL
LIN {X 0,Y 362.604,Z 417.103,A -85,B 0,C 180,E1 17658.456,E2 17658.456} C_VEL
LIN {X 0,Y 361.559,Z 414.752,A -85,B 0,C 180,E1 17656.88,E2 17656.88} C_VEL
LIN {X 0,Y 357.88,Z 409.162,A -85,B 0,C 180,E1 17649.975,E2 17649.975} C_VEL
LIN {X 0,Y 356.873,Z 408.331,A -85,B 0,C 180,E1 17645.305,E2 17645.305} C_VEL
LIN {X 0,Y 357.829,Z 409.002,A -85,B 0,C 180,E1 17640.001,E2 17640.001} C_VEL
LIN {X 0,Y 358.628,Z 410.866,A -85,B 0,C 180,E1 17637.444,E2 17637.444} C_VEL
LIN {X 0,Y 362.414,Z 415.598,A -85,B 0,C 180,E1 17632.072,E2 17632.072} C_VEL
LIN {X 0,Y 364.159,Z 419.177,A -85,B 0,C 180,E1 17629.88,E2 17629.88} C_VEL
LIN {X 0,Y 366.239,Z 421.224,A -85,B 0,C 180,E1 17628.185,E2 17628.185} C_VEL
LIN {X 0,Y 368.192,Z 425.079,A -85,B 0,C 180,E1 17626.335,E2 17626.335} C_VEL
LIN {X 0,Y 369.916,Z 427.116,A -85,B 0,C 180,E1 17625.122,E2 17625.122} C_VEL
LIN {X 0,Y 372.37,Z 431.298,A -85,B 0,C 180,E1 17623.304,E2 17623.304} C_VEL
LIN {X 0,Y 373.56,Z 432.918,A -85,B 0,C 180,E1 17622.556,E2 17622.556} C_VEL
LIN {X 0,Y 376.139,Z 437.056,A -85,B 0,C 180,E1 17620.916,E2 17620.916} C_VEL
LIN {X 0,Y 380.135,Z 443.851,A -85,B 0,C 180,E1 17618.556,E2 17618.556} C_VEL
LIN {X 0,Y 385.136,Z 452.144,A -85,B 0,C 180,E1 17615.947,E2 17615.947} C_VEL
LIN {X 0,Y 392.626,Z 465.719,A -85,B 0,C 180,E1 17612.389,E2 17612.389} C_VEL
LIN {X 0,Y 399.162,Z 475.309,A -85,B 0,C 180,E1 17610.597,E2 17610.597} C_VEL
LIN {X 0,Y 410.014,Z 491.578,A -85,B 0,C 180,E1 17608.01,E2 17608.01} C_VEL
LIN {X 0,Y 416,Z 501.482,A -85,B 0,C 180,E1 17606.673,E2 17606.673} C_VEL
LIN {X 0,Y 416.552,Z 512.636,A -85,B 0,C 180,E1 17606.264,E2 17606.264} C_VEL
LIN {X 0,Y 407.061,Z 702.282,A -85,B 0,C 180,E1 17602.424,E2 17602.424} C_VEL
LIN {X 0,Y 402.042,Z 801.691,A -85,B 0,C 180,E1 17600.353,E2 17600.353} C_VEL
LIN {X 0,Y 399.658,Z 825.247,A -85,B 0,C 180,E1 17599.665,E2 17599.665} C_VEL
LIN {X 0,Y 396.425,Z 849.091,A -85,B 0,C 180,E1 17598.731,E2 17598.731} C_VEL
LIN {X 0,Y 392.999,Z 870.46,A -85,B 0,C 180,E1 17597.643,E2 17597.643} C_VEL
LIN {X 0,Y 388.941,Z 892.394,A -85,B 0,C 180,E1 17596.25,E2 17596.25} C_VEL
LIN {X 0,Y 384.786,Z 913.164,A -85,B 0,C 180,E1 17594.66,E2 17594.66} C_VEL
LIN {X 0,Y 380.228,Z 934.081,A -85,B 0,C 180,E1 17592.723,E2 17592.723} C_VEL
LIN {X 0,Y 375.665,Z 954.367,A -85,B 0,C 180,E1 17590.499,E2 17590.499} C_VEL
LIN {X 0,Y 371.314,Z 973.332,A -85,B 0,C 180,E1 17588.072,E2 17588.072} C_VEL
LIN {X 0,Y 367.186,Z 991.312,A -85,B 0,C 180,E1 17585.355,E2 17585.355} C_VEL
LIN {X 0,Y 363.296,Z 1008.887,A -85,B 0,C 180,E1 17582.271,E2 17582.271} C_VEL
LIN {X 0,Y 360.215,Z 1023.767,A -85,B 0,C 180,E1 17579.244,E2 17579.244} C_VEL
LIN {X 0,Y 357.652,Z 1037.21,A -85,B 0,C 180,E1 17576.035,E2 17576.035} C_VEL
LIN {X 0,Y 355.631,Z 1049.424,A -85,B 0,C 180,E1 17572.655,E2 17572.655} C_VEL
LIN {X 0,Y 354.268,Z 1059.135,A -85,B 0,C 180,E1 17569.453,E2 17569.453} C_VEL
LIN {X 0,Y 353.341,Z 1067.727,A -85,B 0,C 180,E1 17566.1,E2 17566.1} C_VEL
LIN {X 0,Y 352.822,Z 1074.504,A -85,B 0,C 180,E1 17562.77,E2 17562.77} C_VEL
LIN {X 0,Y 352.554,Z 1079.79,A -85,B 0,C 180,E1 17559.468,E2 17559.468} C_VEL
LIN {X 0,Y 352.539,Z 1083.501,A -85,B 0,C 180,E1 17556.024,E2 17556.024} C_VEL
LIN {X 0,Y 352.526,Z 1085.405,A -85,B 0,C 180,E1 17553.089,E2 17553.089} C_VEL
LIN {X 0,Y 352.548,Z 1086.136,A -85,B 0,C 180,E1 17549.837,E2 17549.837} C_VEL
LIN {X 0,Y 352.527,Z 1085.312,A -85,B 0,C 180,E1 17546.711,E2 17546.711} C_VEL
LIN {X 0,Y 352.547,Z 1083.372,A -85,B 0,C 180,E1 17543.813,E2 17543.813} C_VEL
LIN {X 0,Y 352.559,Z 1079.55,A -85,B 0,C 180,E1 17540.368,E2 17540.368} C_VEL
LIN {X 0,Y 352.833,Z 1074.297,A -85,B 0,C 180,E1 17537.114,E2 17537.114} C_VEL
LIN {X 0,Y 353.376,Z 1067.36,A -85,B 0,C 180,E1 17533.733,E2 17533.733} C_VEL
LIN {X 0,Y 354.323,Z 1058.662,A -85,B 0,C 180,E1 17530.378,E2 17530.378} C_VEL
LIN {X 0,Y 355.792,Z 1048.327,A -85,B 0,C 180,E1 17527.007,E2 17527.007} C_VEL
LIN {X 0,Y 357.78,Z 1036.47,A -85,B 0,C 180,E1 17523.775,E2 17523.775} C_VEL
LIN {X 0,Y 360.521,Z 1022.17,A -85,B 0,C 180,E1 17520.418,E2 17520.418} C_VEL
LIN {X 0,Y 363.681,Z 1007.134,A -85,B 0,C 180,E1 17517.394,E2 17517.394} C_VEL
LIN {X 0,Y 367.468,Z 990.048,A -85,B 0,C 180,E1 17514.444,E2 17514.444} C_VEL
LIN {X 0,Y 371.583,Z 972.087,A -85,B 0,C 180,E1 17511.765,E2 17511.765} C_VEL
LIN {X 0,Y 375.846,Z 953.533,A -85,B 0,C 180,E1 17509.405,E2 17509.405} C_VEL
LIN {X 0,Y 380.565,Z 932.436,A -85,B 0,C 180,E1 17507.119,E2 17507.119} C_VEL
LIN {X 0,Y 384.974,Z 912.188,A -85,B 0,C 180,E1 17505.263,E2 17505.263} C_VEL
LIN {X 0,Y 389.149,Z 891.244,A -85,B 0,C 180,E1 17503.674,E2 17503.674} C_VEL
LIN {X 0,Y 393.337,Z 868.206,A -85,B 0,C 180,E1 17502.238,E2 17502.238} C_VEL
LIN {X 0,Y 396.89,Z 845.912,A -85,B 0,C 180,E1 17501.127,E2 17501.127} C_VEL
LIN {X 0,Y 399.92,Z 822.692,A -85,B 0,C 180,E1 17500.255,E2 17500.255} C_VEL
LIN {X 0,Y 402.273,Z 797.421,A -85,B 0,C 180,E1 17499.555,E2 17499.555} C_VEL
LIN {X 0,Y 412.062,Z 601.518,A -85,B 0,C 180,E1 17495.529,E2 17495.529} C_VEL
LIN {X 0,Y 416.486,Z 509.862,A -85,B 0,C 180,E1 17493.663,E2 17493.663} C_VEL
LIN {X 0,Y 415.774,Z 500.914,A -85,B 0,C 180,E1 17493.291,E2 17493.291} C_VEL
LIN {X 0,Y 404.889,Z 483.78,A -85,B 0,C 180,E1 17490.824,E2 17490.824} C_VEL
LIN {X 0,Y 394.057,Z 468.142,A -85,B 0,C 180,E1 17488.119,E2 17488.119} C_VEL
LIN {X 0,Y 391.572,Z 464.039,A -85,B 0,C 180,E1 17487.197,E2 17487.197} C_VEL
LIN {X 0,Y 385.059,Z 452.043,A -85,B 0,C 180,E1 17484.058,E2 17484.058} C_VEL
LIN {X 0,Y 379.022,Z 441.945,A -85,B 0,C 180,E1 17480.862,E2 17480.862} C_VEL
LIN {X 0,Y 375.758,Z 436.638,A -85,B 0,C 180,E1 17478.943,E2 17478.943} C_VEL
LIN {X 0,Y 372.75,Z 431.721,A -85,B 0,C 180,E1 17477,E2 17477} C_VEL
LIN {X 0,Y 369.979,Z 427.353,A -85,B 0,C 180,E1 17475.036,E2 17475.036} C_VEL
LIN {X 0,Y 368.926,Z 425.878,A -85,B 0,C 180,E1 17474.277,E2 17474.277} C_VEL
LIN {X 0,Y 366.635,Z 422.523,A -85,B 0,C 180,E1 17472.441,E2 17472.441} C_VEL
LIN {X 0,Y 365.916,Z 420.873,A -85,B 0,C 180,E1 17471.665,E2 17471.665} C_VEL
LIN {X 0,Y 362.875,Z 417.137,A -85,B 0,C 180,E1 17468.876,E2 17468.876} C_VEL
LIN {X 0,Y 361.991,Z 415.037,A -85,B 0,C 180,E1 17467.618,E2 17467.618} C_VEL
LIN {X 0,Y 358.534,Z 410.59,A -85,B 0,C 180,E1 17462.557,E2 17462.557} C_VEL
LIN {X 0,Y 357.716,Z 408.886,A -85,B 0,C 180,E1 17460.16,E2 17460.16} C_VEL
LIN {X 0,Y 356.682,Z 408.18,A -85,B 0,C 180,E1 17454.53,E2 17454.53} C_VEL
LIN {X 0,Y 357.816,Z 409.069,A -85,B 0,C 180,E1 17449.697,E2 17449.697} C_VEL
LIN {X 0,Y 358.764,Z 411.503,A -85,B 0,C 180,E1 17446.789,E2 17446.789} C_VEL
LIN {X 0,Y 361.968,Z 415.411,A -85,B 0,C 180,E1 17442.31,E2 17442.31} C_VEL
LIN {X 0,Y 363.958,Z 419.316,A -85,B 0,C 180,E1 17439.748,E2 17439.748} C_VEL
LIN {X 0,Y 365.429,Z 420.819,A -85,B 0,C 180,E1 17438.48,E2 17438.48} C_VEL
LIN {X 0,Y 367.424,Z 424.847,A -85,B 0,C 180,E1 17436.42,E2 17436.42} C_VEL
LIN {X 0,Y 368.678,Z 426.29,A -85,B 0,C 180,E1 17435.484,E2 17435.484} C_VEL
LIN {X 0,Y 370.683,Z 430.163,A -85,B 0,C 180,E1 17433.745,E2 17433.745} C_VEL
LIN {X 0,Y 371.911,Z 432.03,A -85,B 0,C 180,E1 17432.858,E2 17432.858} C_VEL
LIN {X 0,Y 374.841,Z 437.253,A -85,B 0,C 180,E1 17430.722,E2 17430.722} C_VEL
LIN {X 0,Y 377.531,Z 442.197,A -85,B 0,C 180,E1 17428.906,E2 17428.906} C_VEL
LIN {X 0,Y 381.817,Z 450.038,A -85,B 0,C 180,E1 17426.278,E2 17426.278} C_VEL
LIN {X 0,Y 387.998,Z 462.606,A -85,B 0,C 180,E1 17422.728,E2 17422.728} C_VEL
LIN {X 0,Y 391.432,Z 469.626,A -85,B 0,C 180,E1 17421.022,E2 17421.022} C_VEL
LIN {X 0,Y 402.6,Z 486.453,A -85,B 0,C 180,E1 17418.201,E2 17418.201} C_VEL
LIN {X 0,Y 408.165,Z 495.714,A -85,B 0,C 180,E1 17416.898,E2 17416.898} C_VEL
LIN {X 0,Y 410.651,Z 516.914,A -85,B 0,C 180,E1 17415.899,E2 17415.899} C_VEL
LIN {X 0,Y 402.208,Z 750.56,A -85,B 0,C 180,E1 17411.738,E2 17411.738} C_VEL
LIN {X 0,Y 400.754,Z 770.964,A -85,B 0,C 180,E1 17411.131,E2 17411.131} C_VEL
LIN {X 0,Y 398.473,Z 791.787,A -85,B 0,C 180,E1 17410.26,E2 17410.26} C_VEL
LIN {X 0,Y 395.625,Z 811.243,A -85,B 0,C 180,E1 17409.185,E2 17409.185} C_VEL
LIN {X 0,Y 392.241,Z 829.669,A -85,B 0,C 180,E1 17407.904,E2 17407.904} C_VEL
LIN {X 0,Y 388.393,Z 847.116,A -85,B 0,C 180,E1 17406.398,E2 17406.398} C_VEL
LIN {X 0,Y 384.026,Z 864.447,A -85,B 0,C 180,E1 17404.583,E2 17404.583} C_VEL
LIN {X 0,Y 379.81,Z 879.664,A -85,B 0,C 180,E1 17402.661,E2 17402.661} C_VEL
LIN {X 0,Y 375.288,Z 894.464,A -85,B 0,C 180,E1 17400.412,E2 17400.412} C_VEL
LIN {X 0,Y 370.974,Z 907.751,A -85,B 0,C 180,E1 17397.968,E2 17397.968} C_VEL
LIN {X 0,Y 366.701,Z 920.449,A -85,B 0,C 180,E1 17395.143,E2 17395.143} C_VEL
LIN {X 0,Y 363.011,Z 931.361,A -85,B 0,C 180,E1 17392.17,E2 17392.17} C_VEL
LIN {X 0,Y 359.993,Z 940.447,A -85,B 0,C 180,E1 17389.132,E2 17389.132} C_VEL
LIN {X 0,Y 357.481,Z 948.42,A -85,B 0,C 180,E1 17385.742,E2 17385.742} C_VEL
LIN {X 0,Y 356.694,Z 950.953,A -85,B 0,C 180,E1 17384.433,E2 17384.433} C_VEL
LIN {X 0,Y 355.124,Z 953.296,A -85,B 0,C 180,E1 17383.268,E2 17383.268} C_VEL
LIN {X 0,Y 347.785,Z 959.134,A -85,B 0,C 180,E1 17380.155,E2 17380.155} C_VEL
LIN {X 0,Y 346.746,Z 960.427,A -85,B 0,C 180,E1 17379.09,E2 17379.09} C_VEL
LIN {X 0,Y 346.042,Z 963.46,A -85,B 0,C 180,E1 17375.472,E2 17375.472} C_VEL
LIN {X 0,Y 345.751,Z 964.978,A -85,B 0,C 180,E1 17371.989,E2 17371.989} C_VEL
LIN {X 0,Y 345.719,Z 965.03,A -85,B 0,C 180,E1 17368.343,E2 17368.343} C_VEL
LIN {X 0,Y 346.009,Z 963.613,A -85,B 0,C 180,E1 17364.694,E2 17364.694} C_VEL
LIN {X 0,Y 346.694,Z 960.67,A -85,B 0,C 180,E1 17361.041,E2 17361.041} C_VEL
LIN {X 0,Y 347.845,Z 956.349,A -85,B 0,C 180,E1 17357.55,E2 17357.55} C_VEL
LIN {X 0,Y 349.712,Z 950.36,A -85,B 0,C 180,E1 17354.069,E2 17354.069} C_VEL
LIN {X 0,Y 352.149,Z 942.905,A -85,B 0,C 180,E1 17350.77,E2 17350.77} C_VEL
LIN {X 0,Y 355.421,Z 933.606,A -85,B 0,C 180,E1 17347.506,E2 17347.506} C_VEL
LIN {X 0,Y 359.277,Z 922.805,A -85,B 0,C 180,E1 17344.446,E2 17344.446} C_VEL
LIN {X 0,Y 363.4,Z 911.249,A -85,B 0,C 180,E1 17341.755,E2 17341.755} C_VEL
LIN {X 0,Y 367.805,Z 898.271,A -85,B 0,C 180,E1 17339.265,E2 17339.265} C_VEL
LIN {X 0,Y 372.425,Z 883.911,A -85,B 0,C 180,E1 17336.975,E2 17336.975} C_VEL
LIN {X 0,Y 377.116,Z 868.094,A -85,B 0,C 180,E1 17334.876,E2 17334.876} C_VEL
LIN {X 0,Y 381.597,Z 851.467,A -85,B 0,C 180,E1 17333.05,E2 17333.05} C_VEL
LIN {X 0,Y 385.77,Z 833.466,A -85,B 0,C 180,E1 17331.439,E2 17331.439} C_VEL
LIN {X 0,Y 389.276,Z 815.689,A -85,B 0,C 180,E1 17330.145,E2 17330.145} C_VEL
LIN {X 0,Y 392.347,Z 796.8,A -85,B 0,C 180,E1 17329.036,E2 17329.036} C_VEL
LIN {X 0,Y 394.794,Z 776.968,A -85,B 0,C 180,E1 17328.138,E2 17328.138} C_VEL
LIN {X 0,Y 396.454,Z 756.525,A -85,B 0,C 180,E1 17327.47,E2 17327.47} C_VEL
LIN {X 0,Y 397.592,Z 730.076,A -85,B 0,C 180,E1 17326.915,E2 17326.915} C_VEL
LIN {X 0,Y 405.73,Z 517.469,A -85,B 0,C 180,E1 17323.122,E2 17323.122} C_VEL
LIN {X 0,Y 403.445,Z 499.653,A -85,B 0,C 180,E1 17322.217,E2 17322.217} C_VEL
LIN {X 0,Y 393.427,Z 483.808,A -85,B 0,C 180,E1 17319.73,E2 17319.73} C_VEL
LIN {X 0,Y 384.762,Z 471.141,A -85,B 0,C 180,E1 17317.358,E2 17317.358} C_VEL
LIN {X 0,Y 382.815,Z 467.942,A -85,B 0,C 180,E1 17316.693,E2 17316.693} C_VEL
LIN {X 0,Y 377.122,Z 456.173,A -85,B 0,C 180,E1 17313.286,E2 17313.286} C_VEL
LIN {X 0,Y 372.046,Z 446.612,A -85,B 0,C 180,E1 17309.992,E2 17309.992} C_VEL
LIN {X 0,Y 369.262,Z 441.648,A -85,B 0,C 180,E1 17308.027,E2 17308.027} C_VEL
LIN {X 0,Y 366.935,Z 437.389,A -85,B 0,C 180,E1 17306.196,E2 17306.196} C_VEL
LIN {X 0,Y 364.689,Z 433.418,A -85,B 0,C 180,E1 17304.284,E2 17304.284} C_VEL
LIN {X 0,Y 361.643,Z 428.286,A -85,B 0,C 180,E1 17301.405,E2 17301.405} C_VEL
LIN {X 0,Y 360.86,Z 427.018,A -85,B 0,C 180,E1 17300.603,E2 17300.603} C_VEL
LIN {X 0,Y 358.586,Z 423.621,A -85,B 0,C 180,E1 17298.03,E2 17298.03} C_VEL
LIN {X 0,Y 357.766,Z 421.761,A -85,B 0,C 180,E1 17296.73,E2 17296.73} C_VEL
LIN {X 0,Y 354.273,Z 416.294,A -85,B 0,C 180,E1 17289.914,E2 17289.914} C_VEL
LIN {X 0,Y 353.359,Z 415.515,A -85,B 0,C 180,E1 17285.196,E2 17285.196} C_VEL
LIN {X 0,Y 354.331,Z 416.204,A -85,B 0,C 180,E1 17280.001,E2 17280.001} C_VEL
LIN {X 0,Y 355.103,Z 417.998,A -85,B 0,C 180,E1 17277.58,E2 17277.58} C_VEL
LIN {X 0,Y 358.8,Z 422.836,A -85,B 0,C 180,E1 17272.152,E2 17272.152} C_VEL
LIN {X 0,Y 360.588,Z 426.337,A -85,B 0,C 180,E1 17269.94,E2 17269.94} C_VEL
LIN {X 0,Y 362.545,Z 428.543,A -85,B 0,C 180,E1 17268.254,E2 17268.254} C_VEL
LIN {X 0,Y 364.603,Z 432.273,A -85,B 0,C 180,E1 17266.359,E2 17266.359} C_VEL
LIN {X 0,Y 365.933,Z 433.745,A -85,B 0,C 180,E1 17265.442,E2 17265.442} C_VEL
LIN {X 0,Y 368.533,Z 438.254,A -85,B 0,C 180,E1 17263.449,E2 17263.449} C_VEL
LIN {X 0,Y 369.661,Z 439.989,A -85,B 0,C 180,E1 17262.691,E2 17262.691} C_VEL
LIN {X 0,Y 372.917,Z 445.415,A -85,B 0,C 180,E1 17260.582,E2 17260.582} C_VEL
LIN {X 0,Y 376.166,Z 450.971,A -85,B 0,C 180,E1 17258.645,E2 17258.645} C_VEL
LIN {X 0,Y 380.587,Z 458.338,A -85,B 0,C 180,E1 17256.3,E2 17256.3} C_VEL
LIN {X 0,Y 385.78,Z 467.59,A -85,B 0,C 180,E1 17253.817,E2 17253.817} C_VEL
LIN {X 0,Y 395.854,Z 481.804,A -85,B 0,C 180,E1 17251.074,E2 17251.074} C_VEL
LIN {X 0,Y 406.36,Z 497.797,A -85,B 0,C 180,E1 17248.497,E2 17248.497} C_VEL
LIN {X 0,Y 411.12,Z 505.865,A -85,B 0,C 180,E1 17247.395,E2 17247.395} C_VEL
LIN {X 0,Y 411.43,Z 514.2,A -85,B 0,C 180,E1 17247.097,E2 17247.097} C_VEL
LIN {X 0,Y 401.552,Z 704.005,A -85,B 0,C 180,E1 17243.226,E2 17243.226} C_VEL
LIN {X 0,Y 396.457,Z 800.948,A -85,B 0,C 180,E1 17241.189,E2 17241.189} C_VEL
LIN {X 0,Y 393.992,Z 824.505,A -85,B 0,C 180,E1 17240.497,E2 17240.497} C_VEL
LIN {X 0,Y 390.59,Z 848.625,A -85,B 0,C 180,E1 17239.546,E2 17239.546} C_VEL
LIN {X 0,Y 386.922,Z 870.59,A -85,B 0,C 180,E1 17238.416,E2 17238.416} C_VEL
LIN {X 0,Y 382.688,Z 892.377,A -85,B 0,C 180,E1 17237.007,E2 17237.007} C_VEL
LIN {X 0,Y 378.174,Z 913.728,A -85,B 0,C 180,E1 17235.334,E2 17235.334} C_VEL
LIN {X 0,Y 373.617,Z 933.682,A -85,B 0,C 180,E1 17233.454,E2 17233.454} C_VEL
LIN {X 0,Y 368.843,Z 953.824,A -85,B 0,C 180,E1 17231.203,E2 17231.203} C_VEL
LIN {X 0,Y 364.285,Z 972.682,A -85,B 0,C 180,E1 17228.741,E2 17228.741} C_VEL
LIN {X 0,Y 359.929,Z 990.652,A -85,B 0,C 180,E1 17225.969,E2 17225.969} C_VEL
LIN {X 0,Y 355.85,Z 1008.051,A -85,B 0,C 180,E1 17222.84,E2 17222.84} C_VEL
LIN {X 0,Y 352.606,Z 1022.872,A -85,B 0,C 180,E1 17219.751,E2 17219.751} C_VEL
LIN {X 0,Y 349.901,Z 1036.233,A -85,B 0,C 180,E1 17216.473,E2 17216.473} C_VEL
LIN {X 0,Y 347.78,Z 1048.369,A -85,B 0,C 180,E1 17213.017,E2 17213.017} C_VEL
LIN {X 0,Y 346.361,Z 1058.045,A -85,B 0,C 180,E1 17209.74,E2 17209.74} C_VEL
LIN {X 0,Y 345.381,Z 1066.933,A -85,B 0,C 180,E1 17206.136,E2 17206.136} C_VEL
LIN {X 0,Y 344.892,Z 1073.317,A -85,B 0,C 180,E1 17202.899,E2 17202.899} C_VEL
LIN {X 0,Y 344.637,Z 1078.763,A -85,B 0,C 180,E1 17199.35,E2 17199.35} C_VEL
LIN {X 0,Y 344.642,Z 1082.237,A -85,B 0,C 180,E1 17195.995,E2 17195.995} C_VEL
LIN {X 0,Y 344.639,Z 1084.109,A -85,B 0,C 180,E1 17192.993,E2 17192.993} C_VEL
LIN {X 0,Y 344.659,Z 1084.745,A -85,B 0,C 180,E1 17189.668,E2 17189.668} C_VEL
LIN {X 0,Y 344.641,Z 1083.949,A -85,B 0,C 180,E1 17186.674,E2 17186.674} C_VEL
LIN {X 0,Y 344.647,Z 1081.963,A -85,B 0,C 180,E1 17183.671,E2 17183.671} C_VEL
LIN {X 0,Y 344.64,Z 1078.331,A -85,B 0,C 180,E1 17180.313,E2 17180.313} C_VEL
LIN {X 0,Y 344.908,Z 1073.016,A -85,B 0,C 180,E1 17176.931,E2 17176.931} C_VEL
LIN {X 0,Y 345.482,Z 1065.828,A -85,B 0,C 180,E1 17173.35,E2 17173.35} C_VEL
LIN {X 0,Y 346.483,Z 1057.095,A -85,B 0,C 180,E1 17169.915,E2 17169.915} C_VEL
LIN {X 0,Y 348.082,Z 1046.464,A -85,B 0,C 180,E1 17166.392,E2 17166.392} C_VEL
LIN {X 0,Y 350.145,Z 1034.911,A -85,B 0,C 180,E1 17163.18,E2 17163.18} C_VEL
LIN {X 0,Y 353.09,Z 1020.477,A -85,B 0,C 180,E1 17159.731,E2 17159.731} C_VEL
LIN {X 0,Y 356.458,Z 1005.424,A -85,B 0,C 180,E1 17156.648,E2 17156.648} C_VEL
LIN {X 0,Y 360.307,Z 989.008,A -85,B 0,C 180,E1 17153.766,E2 17153.766} C_VEL
LIN {X 0,Y 364.718,Z 970.856,A -85,B 0,C 180,E1 17151.011,E2 17151.011} C_VEL
LIN {X 0,Y 369.234,Z 952.153,A -85,B 0,C 180,E1 17148.598,E2 17148.598} C_VEL
LIN {X 0,Y 373.972,Z 932.031,A -85,B 0,C 180,E1 17146.386,E2 17146.386} C_VEL
LIN {X 0,Y 378.779,Z 910.996,A -85,B 0,C 180,E1 17144.435,E2 17144.435} C_VEL
LIN {X 0,Y 382.923,Z 891.119,A -85,B 0,C 180,E1 17142.91,E2 17142.91} C_VEL
LIN {X 0,Y 387.158,Z 868.991,A -85,B 0,C 180,E1 17141.501,E2 17141.501} C_VEL
LIN {X 0,Y 390.703,Z 847.71,A -85,B 0,C 180,E1 17140.417,E2 17140.417} C_VEL
LIN {X 0,Y 394.026,Z 823.904,A -85,B 0,C 180,E1 17139.488,E2 17139.488} C_VEL
LIN {X 0,Y 396.454,Z 800.363,A -85,B 0,C 180,E1 17138.803,E2 17138.803} C_VEL
LIN {X 0,Y 403.242,Z 670.194,A -85,B 0,C 180,E1 17136.081,E2 17136.081} C_VEL
LIN {X 0,Y 411.402,Z 511.535,A -85,B 0,C 180,E1 17132.838,E2 17132.838} C_VEL
LIN {X 0,Y 410.845,Z 505.187,A -85,B 0,C 180,E1 17132.557,E2 17132.557} C_VEL
LIN {X 0,Y 400.364,Z 488.548,A -85,B 0,C 180,E1 17130.089,E2 17130.089} C_VEL
LIN {X 0,Y 389.173,Z 472.24,A -85,B 0,C 180,E1 17127.172,E2 17127.172} C_VEL
LIN {X 0,Y 384.816,Z 466.232,A -85,B 0,C 180,E1 17125.881,E2 17125.881} C_VEL
LIN {X 0,Y 379.343,Z 456.407,A -85,B 0,C 180,E1 17123.124,E2 17123.124} C_VEL
LIN {X 0,Y 374.836,Z 448.574,A -85,B 0,C 180,E1 17120.616,E2 17120.616} C_VEL
LIN {X 0,Y 371.626,Z 443.284,A -85,B 0,C 180,E1 17118.673,E2 17118.673} C_VEL
LIN {X 0,Y 368.674,Z 438.423,A -85,B 0,C 180,E1 17116.706,E2 17116.706} C_VEL
LIN {X 0,Y 365.977,Z 433.973,A -85,B 0,C 180,E1 17114.718,E2 17114.718} C_VEL
LIN {X 0,Y 362.718,Z 429.145,A -85,B 0,C 180,E1 17112.092,E2 17112.092} C_VEL
LIN {X 0,Y 362.131,Z 427.859,A -85,B 0,C 180,E1 17111.466,E2 17111.466} C_VEL
LIN {X 0,Y 359.159,Z 424.071,A -85,B 0,C 180,E1 17108.646,E2 17108.646} C_VEL
LIN {X 0,Y 358.419,Z 422.18,A -85,B 0,C 180,E1 17107.533,E2 17107.533} C_VEL
LIN {X 0,Y 354.97,Z 417.705,A -85,B 0,C 180,E1 17102.421,E2 17102.421} C_VEL
LIN {X 0,Y 354.182,Z 416.07,A -85,B 0,C 180,E1 17100.161,E2 17100.161} C_VEL
LIN {X 0,Y 353.149,Z 415.357,A -85,B 0,C 180,E1 17094.638,E2 17094.638} C_VEL
LIN {X 0,Y 354.196,Z 416.194,A -85,B 0,C 180,E1 17089.755,E2 17089.755} C_VEL
LIN {X 0,Y 355.331,Z 419.08,A -85,B 0,C 180,E1 17086.327,E2 17086.327} C_VEL
LIN {X 0,Y 358.108,Z 422.391,A -85,B 0,C 180,E1 17082.449,E2 17082.449} C_VEL
LIN {X 0,Y 360.083,Z 426.28,A -85,B 0,C 180,E1 17079.859,E2 17079.859} C_VEL
LIN {X 0,Y 361.465,Z 427.867,A -85,B 0,C 180,E1 17078.584,E2 17078.584} C_VEL
LIN {X 0,Y 363.483,Z 431.802,A -85,B 0,C 180,E1 17076.492,E2 17076.492} C_VEL
LIN {X 0,Y 364.643,Z 433.437,A -85,B 0,C 180,E1 17075.54,E2 17075.54} C_VEL
LIN {X 0,Y 366.932,Z 437.399,A -85,B 0,C 180,E1 17073.63,E2 17073.63} C_VEL
LIN {X 0,Y 370.484,Z 443.838,A -85,B 0,C 180,E1 17070.936,E2 17070.936} C_VEL
LIN {X 0,Y 373.412,Z 449.42,A -85,B 0,C 180,E1 17068.883,E2 17068.883} C_VEL
LIN {X 0,Y 377.167,Z 456.346,A -85,B 0,C 180,E1 17066.536,E2 17066.536} C_VEL
LIN {X 0,Y 383.232,Z 468.858,A -85,B 0,C 180,E1 17062.974,E2 17062.974} C_VEL
LIN {X 0,Y 392.744,Z 482.837,A -85,B 0,C 180,E1 17060.329,E2 17060.329} C_VEL
LIN {X 0,Y 402.682,Z 498.418,A -85,B 0,C 180,E1 17057.853,E2 17057.853} C_VEL
LIN {X 0,Y 403.629,Z 500.515,A -85,B 0,C 180,E1 17057.614,E2 17057.614} C_VEL
LIN {X 0,Y 405.637,Z 518.58,A -85,B 0,C 180,E1 17056.755,E2 17056.755} C_VEL
LIN {X 0,Y 396.739,Z 751.276,A -85,B 0,C 180,E1 17052.569,E2 17052.569} C_VEL
LIN {X 0,Y 395.215,Z 771.756,A -85,B 0,C 180,E1 17051.955,E2 17051.955} C_VEL
LIN {X 0,Y 392.911,Z 792.068,A -85,B 0,C 180,E1 17051.102,E2 17051.102} C_VEL
LIN {X 0,Y 390.039,Z 811.198,A -85,B 0,C 180,E1 17050.049,E2 17050.049} C_VEL
LIN {X 0,Y 386.516,Z 829.744,A -85,B 0,C 180,E1 17048.757,E2 17048.757} C_VEL
LIN {X 0,Y 382.515,Z 847.381,A -85,B 0,C 180,E1 17047.238,E2 17047.238} C_VEL
LIN {X 0,Y 377.964,Z 864.866,A -85,B 0,C 180,E1 17045.404,E2 17045.404} C_VEL
LIN {X 0,Y 373.393,Z 880.732,A -85,B 0,C 180,E1 17043.387,E2 17043.387} C_VEL
LIN {X 0,Y 368.827,Z 895.08,A -85,B 0,C 180,E1 17041.184,E2 17041.184} C_VEL
LIN {X 0,Y 364.296,Z 908.477,A -85,B 0,C 180,E1 17038.706,E2 17038.706} C_VEL
LIN {X 0,Y 359.835,Z 921.164,A -85,B 0,C 180,E1 17035.865,E2 17035.865} C_VEL
LIN {X 0,Y 355.953,Z 932.081,A -85,B 0,C 180,E1 17032.876,E2 17032.876} C_VEL
LIN {X 0,Y 352.672,Z 941.437,A -85,B 0,C 180,E1 17029.717,E2 17029.717} C_VEL
LIN {X 0,Y 349.967,Z 949.472,A -85,B 0,C 180,E1 17026.26,E2 17026.26} C_VEL
LIN {X 0,Y 348.02,Z 955.668,A -85,B 0,C 180,E1 17022.781,E2 17022.781} C_VEL
LIN {X 0,Y 346.746,Z 960.427,A -85,B 0,C 180,E1 17019.09,E2 17019.09} C_VEL
LIN {X 0,Y 345.473,Z 961.873,A -85,B 0,C 180,E1 17017.844,E2 17017.844} C_VEL
LIN {X 0,Y 338.667,Z 965.402,A -85,B 0,C 180,E1 17014.417,E2 17014.417} C_VEL
LIN {X 0,Y 337.939,Z 965.896,A -85,B 0,C 180,E1 17013.389,E2 17013.389} C_VEL
LIN {X 0,Y 337.824,Z 966.564,A -85,B 0,C 180,E1 17009.83,E2 17009.83} C_VEL
LIN {X 0,Y 337.981,Z 965.762,A -85,B 0,C 180,E1 17006.098,E2 17006.098} C_VEL
LIN {X 0,Y 338.531,Z 963.441,A -85,B 0,C 180,E1 17002.362,E2 17002.362} C_VEL
LIN {X 0,Y 339.558,Z 959.543,A -85,B 0,C 180,E1 16998.622,E2 16998.622} C_VEL
LIN {X 0,Y 341.239,Z 954.212,A -85,B 0,C 180,E1 16995.058,E2 16995.058} C_VEL
LIN {X 0,Y 343.678,Z 947.15,A -85,B 0,C 180,E1 16991.511,E2 16991.511} C_VEL
LIN {X 0,Y 347.019,Z 938.081,A -85,B 0,C 180,E1 16988.002,E2 16988.002} C_VEL
LIN {X 0,Y 350.796,Z 927.902,A -85,B 0,C 180,E1 16984.869,E2 16984.869} C_VEL
LIN {X 0,Y 355.142,Z 916.279,A -85,B 0,C 180,E1 16981.955,E2 16981.955} C_VEL
LIN {X 0,Y 359.86,Z 903.205,A -85,B 0,C 180,E1 16979.253,E2 16979.253} C_VEL
LIN {X 0,Y 364.722,Z 889.11,A -85,B 0,C 180,E1 16976.844,E2 16976.844} C_VEL
LIN {X 0,Y 369.492,Z 873.956,A -85,B 0,C 180,E1 16974.708,E2 16974.708} C_VEL
LIN {X 0,Y 374.074,Z 857.977,A -85,B 0,C 180,E1 16972.838,E2 16972.838} C_VEL
LIN {X 0,Y 378.493,Z 840.667,A -85,B 0,C 180,E1 16971.158,E2 16971.158} C_VEL
LIN {X 0,Y 382.537,Z 822.14,A -85,B 0,C 180,E1 16969.691,E2 16969.691} C_VEL
LIN {X 0,Y 385.805,Z 803.764,A -85,B 0,C 180,E1 16968.535,E2 16968.535} C_VEL
LIN {X 0,Y 388.662,Z 783.355,A -85,B 0,C 180,E1 16967.529,E2 16967.529} C_VEL
LIN {X 0,Y 390.646,Z 763.492,A -85,B 0,C 180,E1 16966.796,E2 16966.796} C_VEL
LIN {X 0,Y 391.818,Z 742.835,A -85,B 0,C 180,E1 16966.278,E2 16966.278} C_VEL
LIN {X 0,Y 400.8,Z 518.898,A -85,B 0,C 180,E1 16962.234,E2 16962.234} C_VEL
LIN {X 0,Y 398.952,Z 504.221,A -85,B 0,C 180,E1 16961.469,E2 16961.469} C_VEL
LIN {X 0,Y 388.545,Z 487.615,A -85,B 0,C 180,E1 16958.771,E2 16958.771} C_VEL
LIN {X 0,Y 378.618,Z 473.196,A -85,B 0,C 180,E1 16955.893,E2 16955.893} C_VEL
LIN {X 0,Y 374.959,Z 467.715,A -85,B 0,C 180,E1 16954.61,E2 16954.61} C_VEL
LIN {X 0,Y 370.306,Z 458.146,A -85,B 0,C 180,E1 16951.589,E2 16951.589} C_VEL
LIN {X 0,Y 365.376,Z 448.816,A -85,B 0,C 180,E1 16948.079,E2 16948.079} C_VEL
LIN {X 0,Y 362.506,Z 443.815,A -85,B 0,C 180,E1 16945.836,E2 16945.836} C_VEL
LIN {X 0,Y 359.966,Z 439.197,A -85,B 0,C 180,E1 16943.561,E2 16943.561} C_VEL
LIN {X 0,Y 357.587,Z 434.984,A -85,B 0,C 180,E1 16941.144,E2 16941.144} C_VEL
LIN {X 0,Y 356.602,Z 433.645,A -85,B 0,C 180,E1 16940.175,E2 16940.175} C_VEL
LIN {X 0,Y 354.556,Z 430.079,A -85,B 0,C 180,E1 16937.563,E2 16937.563} C_VEL
LIN {X 0,Y 353.827,Z 428.656,A -85,B 0,C 180,E1 16936.415,E2 16936.415} C_VEL
LIN {X 0,Y 350.651,Z 423.419,A -85,B 0,C 180,E1 16929.851,E2 16929.851} C_VEL
LIN {X 0,Y 349.834,Z 422.694,A -85,B 0,C 180,E1 16925.084,E2 16925.084} C_VEL
LIN {X 0,Y 350.847,Z 423.414,A -85,B 0,C 180,E1 16920.001,E2 16920.001} C_VEL
LIN {X 0,Y 351.591,Z 425.273,A -85,B 0,C 180,E1 16917.556,E2 16917.556} C_VEL
LIN {X 0,Y 355.107,Z 429.776,A -85,B 0,C 180,E1 16912.396,E2 16912.396} C_VEL
LIN {X 0,Y 356.822,Z 433.287,A -85,B 0,C 180,E1 16910.159,E2 16910.159} C_VEL
LIN {X 0,Y 358.672,Z 435.226,A -85,B 0,C 180,E1 16908.585,E2 16908.585} C_VEL
LIN {X 0,Y 360.795,Z 439.218,A -85,B 0,C 180,E1 16906.539,E2 16906.539} C_VEL
LIN {X 0,Y 362.066,Z 440.775,A -85,B 0,C 180,E1 16905.61,E2 16905.61} C_VEL
LIN {X 0,Y 364.933,Z 445.479,A -85,B 0,C 180,E1 16903.445,E2 16903.445} C_VEL
LIN {X 0,Y 368.758,Z 452.038,A -85,B 0,C 180,E1 16900.848,E2 16900.848} C_VEL
LIN {X 0,Y 372.041,Z 457.753,A -85,B 0,C 180,E1 16898.839,E2 16898.839} C_VEL
LIN {X 0,Y 376.612,Z 465.636,A -85,B 0,C 180,E1 16896.339,E2 16896.339} C_VEL
LIN {X 0,Y 380.076,Z 470.77,A -85,B 0,C 180,E1 16895.109,E2 16895.109} C_VEL
LIN {X 0,Y 388.531,Z 482.363,A -85,B 0,C 180,E1 16892.655,E2 16892.655} C_VEL
LIN {X 0,Y 399.085,Z 498.185,A -85,B 0,C 180,E1 16889.888,E2 16889.888} C_VEL
LIN {X 0,Y 406.295,Z 510.133,A -85,B 0,C 180,E1 16888.139,E2 16888.139} C_VEL
LIN {X 0,Y 406.385,Z 516.023,A -85,B 0,C 180,E1 16887.945,E2 16887.945} C_VEL
LIN {X 0,Y 396.092,Z 706.366,A -85,B 0,C 180,E1 16884.038,E2 16884.038} C_VEL
LIN {X 0,Y 390.954,Z 800.346,A -85,B 0,C 180,E1 16882.047,E2 16882.047} C_VEL
LIN {X 0,Y 388.401,Z 823.902,A -85,B 0,C 180,E1 16881.35,E2 16881.35} C_VEL
LIN {X 0,Y 384.839,Z 848.183,A -85,B 0,C 180,E1 16880.385,E2 16880.385} C_VEL
LIN {X 0,Y 380.919,Z 870.733,A -85,B 0,C 180,E1 16879.213,E2 16879.213} C_VEL
LIN {X 0,Y 376.511,Z 892.359,A -85,B 0,C 180,E1 16877.79,E2 16877.79} C_VEL
LIN {X 0,Y 371.654,Z 914.16,A -85,B 0,C 180,E1 16876.046,E2 16876.046} C_VEL
LIN {X 0,Y 366.706,Z 934.889,A -85,B 0,C 180,E1 16874.05,E2 16874.05} C_VEL
LIN {X 0,Y 361.744,Z 954.63,A -85,B 0,C 180,E1 16871.769,E2 16871.769} C_VEL
LIN {X 0,Y 356.706,Z 974.277,A -85,B 0,C 180,E1 16869.101,E2 16869.101} C_VEL
LIN {X 0,Y 352.235,Z 991.984,A -85,B 0,C 180,E1 16866.278,E2 16866.278} C_VEL
LIN {X 0,Y 348.23,Z 1008.104,A -85,B 0,C 180,E1 16863.258,E2 16863.258} C_VEL
LIN {X 0,Y 344.688,Z 1023.43,A -85,B 0,C 180,E1 16859.93,E2 16859.93} C_VEL
LIN {X 0,Y 341.923,Z 1036.6,A -85,B 0,C 180,E1 16856.578,E2 16856.578} C_VEL
LIN {X 0,Y 339.697,Z 1048.877,A -85,B 0,C 180,E1 16852.888,E2 16852.888} C_VEL
LIN {X 0,Y 338.231,Z 1058.878,A -85,B 0,C 180,E1 16849.335,E2 16849.335} C_VEL
LIN {X 0,Y 337.346,Z 1066.885,A -85,B 0,C 180,E1 16845.824,E2 16845.824} C_VEL
LIN {X 0,Y 336.893,Z 1073.368,A -85,B 0,C 180,E1 16842.339,E2 16842.339} C_VEL
LIN {X 0,Y 336.734,Z 1078.323,A -85,B 0,C 180,E1 16838.71,E2 16838.71} C_VEL
LIN {X 0,Y 336.733,Z 1081.254,A -85,B 0,C 180,E1 16835.623,E2 16835.623} C_VEL
LIN {X 0,Y 336.781,Z 1083.075,A -85,B 0,C 180,E1 16832.212,E2 16832.212} C_VEL
LIN {X 0,Y 336.778,Z 1083.276,A -85,B 0,C 180,E1 16828.979,E2 16828.979} C_VEL
LIN {X 0,Y 336.769,Z 1082.287,A -85,B 0,C 180,E1 16825.999,E2 16825.999} C_VEL
LIN {X 0,Y 336.71,Z 1079.663,A -85,B 0,C 180,E1 16822.492,E2 16822.492} C_VEL
LIN {X 0,Y 336.792,Z 1075.422,A -85,B 0,C 180,E1 16819.047,E2 16819.047} C_VEL
LIN {X 0,Y 337.083,Z 1070.022,A -85,B 0,C 180,E1 16815.747,E2 16815.747} C_VEL
LIN {X 0,Y 337.823,Z 1062.238,A -85,B 0,C 180,E1 16812.073,E2 16812.073} C_VEL
LIN {X 0,Y 339.031,Z 1053.172,A -85,B 0,C 180,E1 16808.549,E2 16808.549} C_VEL
LIN {X 0,Y 340.873,Z 1042.118,A -85,B 0,C 180,E1 16805.007,E2 16805.007} C_VEL
LIN {X 0,Y 343.432,Z 1029.236,A -85,B 0,C 180,E1 16801.48,E2 16801.48} C_VEL
LIN {X 0,Y 346.632,Z 1014.828,A -85,B 0,C 180,E1 16798.138,E2 16798.138} C_VEL
LIN {X 0,Y 350.471,Z 998.847,A -85,B 0,C 180,E1 16794.962,E2 16794.962} C_VEL
LIN {X 0,Y 354.874,Z 981.543,A -85,B 0,C 180,E1 16792.002,E2 16792.002} C_VEL
LIN {X 0,Y 359.591,Z 962.923,A -85,B 0,C 180,E1 16789.304,E2 16789.304} C_VEL
LIN {X 0,Y 364.747,Z 942.659,A -85,B 0,C 180,E1 16786.816,E2 16786.816} C_VEL
LIN {X 0,Y 369.612,Z 922.914,A -85,B 0,C 180,E1 16784.756,E2 16784.756} C_VEL
LIN {X 0,Y 374.439,Z 901.66,A -85,B 0,C 180,E1 16782.915,E2 16782.915} C_VEL
LIN {X 0,Y 379.257,Z 878.775,A -85,B 0,C 180,E1 16781.291,E2 16781.291} C_VEL
LIN {X 0,Y 383.449,Z 856.528,A -85,B 0,C 180,E1 16780.018,E2 16780.018} C_VEL
LIN {X 0,Y 386.857,Z 834.89,A -85,B 0,C 180,E1 16779.058,E2 16779.058} C_VEL
LIN {X 0,Y 389.988,Z 809.997,A -85,B 0,C 180,E1 16778.226,E2 16778.226} C_VEL
LIN {X 0,Y 391.857,Z 786.039,A -85,B 0,C 180,E1 16777.631,E2 16777.631} C_VEL
LIN {X 0,Y 402.849,Z 580.137,A -85,B 0,C 180,E1 16773.36,E2 16773.36} C_VEL
LIN {X 0,Y 406.363,Z 512.495,A -85,B 0,C 180,E1 16771.964,E2 16771.964} C_VEL
LIN {X 0,Y 406.07,Z 509.57,A -85,B 0,C 180,E1 16771.823,E2 16771.823} C_VEL
LIN {X 0,Y 395.65,Z 492.997,A -85,B 0,C 180,E1 16769.274,E2 16769.274} C_VEL
LIN {X 0,Y 385.519,Z 478.187,A -85,B 0,C 180,E1 16766.534,E2 16766.534} C_VEL
LIN {X 0,Y 377.054,Z 466.523,A -85,B 0,C 180,E1 16763.936,E2 16763.936} C_VEL
LIN {X 0,Y 372.652,Z 458.849,A -85,B 0,C 180,E1 16761.566,E2 16761.566} C_VEL
LIN {X 0,Y 369.854,Z 454.067,A -85,B 0,C 180,E1 16759.914,E2 16759.914} C_VEL
LIN {X 0,Y 367.472,Z 449.911,A -85,B 0,C 180,E1 16758.398,E2 16758.398} C_VEL
LIN {X 0,Y 364.571,Z 445.09,A -85,B 0,C 180,E1 16756.408,E2 16756.408} C_VEL
LIN {X 0,Y 361.556,Z 440.028,A -85,B 0,C 180,E1 16754.084,E2 16754.084} C_VEL
LIN {X 0,Y 359.074,Z 436.46,A -85,B 0,C 180,E1 16752.054,E2 16752.054} C_VEL
LIN {X 0,Y 358.352,Z 434.841,A -85,B 0,C 180,E1 16751.262,E2 16751.262} C_VEL
LIN {X 0,Y 355.44,Z 431,A -85,B 0,C 180,E1 16748.411,E2 16748.411} C_VEL
LIN {X 0,Y 354.682,Z 429.205,A -85,B 0,C 180,E1 16747.287,E2 16747.287} C_VEL
LIN {X 0,Y 351.367,Z 424.647,A -85,B 0,C 180,E1 16742.12,E2 16742.12} C_VEL
LIN {X 0,Y 350.56,Z 423.184,A -85,B 0,C 180,E1 16739.836,E2 16739.836} C_VEL
LIN {X 0,Y 349.644,Z 422.539,A -85,B 0,C 180,E1 16734.255,E2 16734.255} C_VEL
LIN {X 0,Y 350.629,Z 423.391,A -85,B 0,C 180,E1 16729.65,E2 16729.65} C_VEL
LIN {X 0,Y 354.261,Z 429.38,A -85,B 0,C 180,E1 16722.592,E2 16722.592} C_VEL
LIN {X 0,Y 356.2,Z 433.238,A -85,B 0,C 180,E1 16719.973,E2 16719.973} C_VEL
LIN {X 0,Y 357.53,Z 434.929,A -85,B 0,C 180,E1 16718.681,E2 16718.681} C_VEL
LIN {X 0,Y 359.751,Z 438.989,A -85,B 0,C 180,E1 16716.408,E2 16716.408} C_VEL
LIN {X 0,Y 360.631,Z 440.541,A -85,B 0,C 180,E1 16715.599,E2 16715.599} C_VEL
LIN {X 0,Y 363.507,Z 445.603,A -85,B 0,C 180,E1 16713.185,E2 16713.185} C_VEL
LIN {X 0,Y 366.208,Z 450.574,A -85,B 0,C 180,E1 16711.101,E2 16711.101} C_VEL
LIN {X 0,Y 368.872,Z 455.716,A -85,B 0,C 180,E1 16709.182,E2 16709.182} C_VEL
LIN {X 0,Y 372.525,Z 462.653,A -85,B 0,C 180,E1 16706.801,E2 16706.801} C_VEL
LIN {X 0,Y 375.879,Z 469.424,A -85,B 0,C 180,E1 16704.837,E2 16704.837} C_VEL
LIN {X 0,Y 384.85,Z 482.143,A -85,B 0,C 180,E1 16702.136,E2 16702.136} C_VEL
LIN {X 0,Y 395.15,Z 498.127,A -85,B 0,C 180,E1 16699.364,E2 16699.364} C_VEL
LIN {X 0,Y 399.11,Z 504.869,A -85,B 0,C 180,E1 16698.37,E2 16698.37} C_VEL
LIN {X 0,Y 400.722,Z 520.133,A -85,B 0,C 180,E1 16697.635,E2 16697.635} C_VEL
LIN {X 0,Y 391.355,Z 751.927,A -85,B 0,C 180,E1 16693.424,E2 16693.424} C_VEL
LIN {X 0,Y 389.767,Z 772.435,A -85,B 0,C 180,E1 16692.805,E2 16692.805} C_VEL
LIN {X 0,Y 387.286,Z 793.4,A -85,B 0,C 180,E1 16691.915,E2 16691.915} C_VEL
LIN {X 0,Y 384.335,Z 812.237,A -85,B 0,C 180,E1 16690.866,E2 16690.866} C_VEL
LIN {X 0,Y 380.682,Z 830.775,A -85,B 0,C 180,E1 16689.563,E2 16689.563} C_VEL
LIN {X 0,Y 376.528,Z 848.408,A -85,B 0,C 180,E1 16688.03,E2 16688.03} C_VEL
LIN {X 0,Y 371.801,Z 865.905,A -85,B 0,C 180,E1 16686.178,E2 16686.178} C_VEL
LIN {X 0,Y 367.036,Z 881.792,A -85,B 0,C 180,E1 16684.137,E2 16684.137} C_VEL
LIN {X 0,Y 362.127,Z 896.629,A -85,B 0,C 180,E1 16681.828,E2 16681.828} C_VEL
LIN {X 0,Y 357.402,Z 909.972,A -85,B 0,C 180,E1 16679.313,E2 16679.313} C_VEL
LIN {X 0,Y 352.672,Z 922.811,A -85,B 0,C 180,E1 16676.376,E2 16676.376} C_VEL
LIN {X 0,Y 348.595,Z 933.712,A -85,B 0,C 180,E1 16673.317,E2 16673.317} C_VEL
LIN {X 0,Y 345.227,Z 942.854,A -85,B 0,C 180,E1 16670.161,E2 16670.161} C_VEL
LIN {X 0,Y 342.367,Z 950.875,A -85,B 0,C 180,E1 16666.631,E2 16666.631} C_VEL
LIN {X 0,Y 340.302,Z 957.056,A -85,B 0,C 180,E1 16663.076,E2 16663.076} C_VEL
LIN {X 0,Y 338.948,Z 961.767,A -85,B 0,C 180,E1 16659.337,E2 16659.337} C_VEL
LIN {X 0,Y 338.183,Z 964.829,A -85,B 0,C 180,E1 16655.599,E2 16655.599} C_VEL
LIN {X 0,Y 337.939,Z 965.896,A -85,B 0,C 180,E1 16653.389,E2 16653.389} C_VEL
LIN {X 0,Y 336.88,Z 966.505,A -85,B 0,C 180,E1 16652.087,E2 16652.087} C_VEL
LIN {X 0,Y 330.605,Z 967.746,A -85,B 0,C 180,E1 16648.498,E2 16648.498} C_VEL
LIN {X 0,Y 330.008,Z 967.593,A -85,B 0,C 180,E1 16647.439,E2 16647.439} C_VEL
LIN {X 0,Y 330.427,Z 965.881,A -85,B 0,C 180,E1 16643.572,E2 16643.572} C_VEL
LIN {X 0,Y 331.338,Z 962.549,A -85,B 0,C 180,E1 16639.744,E2 16639.744} C_VEL
LIN {X 0,Y 332.874,Z 957.642,A -85,B 0,C 180,E1 16635.979,E2 16635.979} C_VEL
LIN {X 0,Y 335.213,Z 951.064,A -85,B 0,C 180,E1 16632.287,E2 16632.287} C_VEL
LIN {X 0,Y 338.23,Z 943.164,A -85,B 0,C 180,E1 16628.86,E2 16628.86} C_VEL
LIN {X 0,Y 342.104,Z 933.347,A -85,B 0,C 180,E1 16625.479,E2 16625.479} C_VEL
LIN {X 0,Y 346.348,Z 922.522,A -85,B 0,C 180,E1 16622.49,E2 16622.49} C_VEL
LIN {X 0,Y 351.001,Z 910.344,A -85,B 0,C 180,E1 16619.721,E2 16619.721} C_VEL
LIN {X 0,Y 355.986,Z 896.809,A -85,B 0,C 180,E1 16617.174,E2 16617.174} C_VEL
LIN {X 0,Y 361.133,Z 881.842,A -85,B 0,C 180,E1 16614.838,E2 16614.838} C_VEL
LIN {X 0,Y 366.136,Z 865.736,A -85,B 0,C 180,E1 16612.779,E2 16612.779} C_VEL
LIN {X 0,Y 370.858,Z 848.721,A -85,B 0,C 180,E1 16610.984,E2 16610.984} C_VEL
LIN {X 0,Y 375.248,Z 830.548,A -85,B 0,C 180,E1 16609.411,E2 16609.411} C_VEL
LIN {X 0,Y 379.117,Z 811.474,A -85,B 0,C 180,E1 16608.077,E2 16608.077} C_VEL
LIN {X 0,Y 382.259,Z 791.644,A -85,B 0,C 180,E1 16606.997,E2 16606.997} C_VEL
LIN {X 0,Y 384.628,Z 771.534,A -85,B 0,C 180,E1 16606.168,E2 16606.168} C_VEL
LIN {X 0,Y 386.212,Z 750.556,A -85,B 0,C 180,E1 16605.553,E2 16605.553} C_VEL
LIN {X 0,Y 395.946,Z 520.137,A -85,B 0,C 180,E1 16601.315,E2 16601.315} C_VEL
LIN {X 0,Y 394.568,Z 508.951,A -85,B 0,C 180,E1 16600.716,E2 16600.716} C_VEL
LIN {X 0,Y 385.078,Z 493.673,A -85,B 0,C 180,E1 16598.168,E2 16598.168} C_VEL
LIN {X 0,Y 375.944,Z 480.115,A -85,B 0,C 180,E1 16595.436,E2 16595.436} C_VEL
LIN {X 0,Y 367.438,Z 468.04,A -85,B 0,C 180,E1 16592.481,E2 16592.481} C_VEL
LIN {X 0,Y 363.014,Z 459.254,A -85,B 0,C 180,E1 16589.359,E2 16589.359} C_VEL
LIN {X 0,Y 360.475,Z 454.523,A -85,B 0,C 180,E1 16587.416,E2 16587.416} C_VEL
LIN {X 0,Y 358.337,Z 450.523,A -85,B 0,C 180,E1 16585.626,E2 16585.626} C_VEL
LIN {X 0,Y 355.867,Z 445.962,A -85,B 0,C 180,E1 16583.339,E2 16583.339} C_VEL
LIN {X 0,Y 353.531,Z 441.679,A -85,B 0,C 180,E1 16580.877,E2 16580.877} C_VEL
LIN {X 0,Y 350.71,Z 437.061,A -85,B 0,C 180,E1 16577.419,E2 16577.419} C_VEL
LIN {X 0,Y 350.033,Z 435.68,A -85,B 0,C 180,E1 16576.305,E2 16576.305} C_VEL
LIN {X 0,Y 347.049,Z 430.553,A -85,B 0,C 180,E1 16569.787,E2 16569.787} C_VEL
LIN {X 0,Y 346.317,Z 429.87,A -85,B 0,C 180,E1 16564.803,E2 16564.803} C_VEL
LIN {X 0,Y 347.412,Z 430.704,A -85,B 0,C 180,E1 16559.836,E2 16559.836} C_VEL
LIN {X 0,Y 348.782,Z 433.853,A -85,B 0,C 180,E1 16556.055,E2 16556.055} C_VEL
LIN {X 0,Y 351.405,Z 436.708,A -85,B 0,C 180,E1 16552.644,E2 16552.644} C_VEL
LIN {X 0,Y 353.228,Z 440.435,A -85,B 0,C 180,E1 16550.222,E2 16550.222} C_VEL
LIN {X 0,Y 354.978,Z 442.555,A -85,B 0,C 180,E1 16548.629,E2 16548.629} C_VEL
LIN {X 0,Y 357.4,Z 446.631,A -85,B 0,C 180,E1 16546.409,E2 16546.409} C_VEL
LIN {X 0,Y 358.521,Z 448.543,A -85,B 0,C 180,E1 16545.464,E2 16545.464} C_VEL
LIN {X 0,Y 361.659,Z 453.644,A -85,B 0,C 180,E1 16543.125,E2 16543.125} C_VEL
LIN {X 0,Y 364.644,Z 458.755,A -85,B 0,C 180,E1 16541.085,E2 16541.085} C_VEL
LIN {X 0,Y 369.669,Z 467.223,A -85,B 0,C 180,E1 16538.126,E2 16538.126} C_VEL
LIN {X 0,Y 379.909,Z 481.094,A -85,B 0,C 180,E1 16534.764,E2 16534.764} C_VEL
LIN {X 0,Y 389.091,Z 494.425,A -85,B 0,C 180,E1 16532.116,E2 16532.116} C_VEL
LIN {X 0,Y 399.138,Z 510.232,A -85,B 0,C 180,E1 16529.498,E2 16529.498} C_VEL
LIN {X 0,Y 401.559,Z 514.733,A -85,B 0,C 180,E1 16528.887,E2 16528.887} C_VEL
LIN {X 0,Y 391.683,Z 691.316,A -85,B 0,C 180,E1 16525.236,E2 16525.236} C_VEL
LIN {X 0,Y 385.586,Z 799.154,A -85,B 0,C 180,E1 16522.942,E2 16522.942} C_VEL
LIN {X 0,Y 383.003,Z 822.569,A -85,B 0,C 180,E1 16522.251,E2 16522.251} C_VEL
LIN {X 0,Y 379.463,Z 846.043,A -85,B 0,C 180,E1 16521.332,E2 16521.332} C_VEL
LIN {X 0,Y 375.493,Z 868.111,A -85,B 0,C 180,E1 16520.194,E2 16520.194} C_VEL
LIN {X 0,Y 371.152,Z 888.921,A -85,B 0,C 180,E1 16518.847,E2 16518.847} C_VEL
LIN {X 0,Y 366.343,Z 910.09,A -85,B 0,C 180,E1 16517.189,E2 16517.189} C_VEL
LIN {X 0,Y 361.402,Z 929.783,A -85,B 0,C 180,E1 16515.318,E2 16515.318} C_VEL
LIN {X 0,Y 355.911,Z 950.805,A -85,B 0,C 180,E1 16512.942,E2 16512.942} C_VEL
LIN {X 0,Y 350.893,Z 969.648,A -85,B 0,C 180,E1 16510.422,E2 16510.422} C_VEL
LIN {X 0,Y 345.985,Z 987.619,A -85,B 0,C 180,E1 16507.573,E2 16507.573} C_VEL
LIN {X 0,Y 341.406,Z 1005.1,A -85,B 0,C 180,E1 16504.323,E2 16504.323} C_VEL
LIN {X 0,Y 337.644,Z 1020.347,A -85,B 0,C 180,E1 16501.015,E2 16501.015} C_VEL
LIN {X 0,Y 334.604,Z 1033.68,A -85,B 0,C 180,E1 16497.592,E2 16497.592} C_VEL
LIN {X 0,Y 332.117,Z 1046.321,A -85,B 0,C 180,E1 16493.792,E2 16493.792} C_VEL
LIN {X 0,Y 330.638,Z 1055.456,A -85,B 0,C 180,E1 16490.536,E2 16490.536} C_VEL
LIN {X 0,Y 329.553,Z 1064.321,A -85,B 0,C 180,E1 16486.752,E2 16486.752} C_VEL
LIN {X 0,Y 329.04,Z 1070.708,A -85,B 0,C 180,E1 16483.353,E2 16483.353} C_VEL
LIN {X 0,Y 328.798,Z 1076.127,A -85,B 0,C 180,E1 16479.628,E2 16479.628} C_VEL
LIN {X 0,Y 328.843,Z 1079.457,A -85,B 0,C 180,E1 16476.284,E2 16476.284} C_VEL
LIN {X 0,Y 328.864,Z 1081.364,A -85,B 0,C 180,E1 16473.137,E2 16473.137} C_VEL
LIN {X 0,Y 328.893,Z 1082.014,A -85,B 0,C 180,E1 16469.652,E2 16469.652} C_VEL
LIN {X 0,Y 328.868,Z 1081.202,A -85,B 0,C 180,E1 16466.514,E2 16466.514} C_VEL
LIN {X 0,Y 328.83,Z 1079.316,A -85,B 0,C 180,E1 16463.54,E2 16463.54} C_VEL
LIN {X 0,Y 328.804,Z 1075.72,A -85,B 0,C 180,E1 16460.018,E2 16460.018} C_VEL
LIN {X 0,Y 329.055,Z 1070.403,A -85,B 0,C 180,E1 16456.469,E2 16456.469} C_VEL
LIN {X 0,Y 329.635,Z 1063.481,A -85,B 0,C 180,E1 16452.834,E2 16452.834} C_VEL
LIN {X 0,Y 330.783,Z 1054.502,A -85,B 0,C 180,E1 16449.103,E2 16449.103} C_VEL
LIN {X 0,Y 332.536,Z 1044.142,A -85,B 0,C 180,E1 16445.485,E2 16445.485} C_VEL
LIN {X 0,Y 334.889,Z 1032.354,A -85,B 0,C 180,E1 16442.047,E2 16442.047} C_VEL
LIN {X 0,Y 338.185,Z 1017.954,A -85,B 0,C 180,E1 16438.445,E2 16438.445} C_VEL
LIN {X 0,Y 341.965,Z 1002.93,A -85,B 0,C 180,E1 16435.239,E2 16435.239} C_VEL
LIN {X 0,Y 346.394,Z 986.041,A -85,B 0,C 180,E1 16432.165,E2 16432.165} C_VEL
LIN {X 0,Y 351.332,Z 967.84,A -85,B 0,C 180,E1 16429.329,E2 16429.329} C_VEL
LIN {X 0,Y 356.383,Z 949.002,A -85,B 0,C 180,E1 16426.839,E2 16426.839} C_VEL
LIN {X 0,Y 361.54,Z 929.135,A -85,B 0,C 180,E1 16424.623,E2 16424.623} C_VEL
LIN {X 0,Y 366.583,Z 908.945,A -85,B 0,C 180,E1 16422.72,E2 16422.72} C_VEL
LIN {X 0,Y 371.419,Z 887.535,A -85,B 0,C 180,E1 16421.059,E2 16421.059} C_VEL
LIN {X 0,Y 376.066,Z 864.739,A -85,B 0,C 180,E1 16419.624,E2 16419.624} C_VEL
LIN {X 0,Y 380.01,Z 842.66,A -85,B 0,C 180,E1 16418.518,E2 16418.518} C_VEL
LIN {X 0,Y 383.387,Z 819.328,A -85,B 0,C 180,E1 16417.649,E2 16417.649} C_VEL
LIN {X 0,Y 385.859,Z 794.506,A -85,B 0,C 180,E1 16416.956,E2 16416.956} C_VEL
LIN {X 0,Y 396.72,Z 600.625,A -85,B 0,C 180,E1 16412.887,E2 16412.887} C_VEL
LIN {X 0,Y 401.449,Z 514.231,A -85,B 0,C 180,E1 16411.097,E2 16411.097} C_VEL
LIN {X 0,Y 391.389,Z 497.957,A -85,B 0,C 180,E1 16408.536,E2 16408.536} C_VEL
LIN {X 0,Y 381.918,Z 484.104,A -85,B 0,C 180,E1 16405.883,E2 16405.883} C_VEL
LIN {X 0,Y 372.906,Z 471.585,A -85,B 0,C 180,E1 16403.045,E2 16403.045} C_VEL
LIN {X 0,Y 369.003,Z 466.33,A -85,B 0,C 180,E1 16401.623,E2 16401.623} C_VEL
LIN {X 0,Y 365.42,Z 460.274,A -85,B 0,C 180,E1 16399.5,E2 16399.5} C_VEL
LIN {X 0,Y 363.329,Z 456.536,A -85,B 0,C 180,E1 16398.117,E2 16398.117} C_VEL
LIN {X 0,Y 360.714,Z 452.034,A -85,B 0,C 180,E1 16396.257,E2 16396.257} C_VEL
LIN {X 0,Y 357.495,Z 446.743,A -85,B 0,C 180,E1 16393.752,E2 16393.752} C_VEL
LIN {X 0,Y 354.996,Z 442.717,A -85,B 0,C 180,E1 16391.535,E2 16391.535} C_VEL
LIN {X 0,Y 354.163,Z 441.457,A -85,B 0,C 180,E1 16390.738,E2 16390.738} C_VEL
LIN {X 0,Y 351.624,Z 437.649,A -85,B 0,C 180,E1 16388.009,E2 16388.009} C_VEL
LIN {X 0,Y 351.113,Z 436.348,A -85,B 0,C 180,E1 16387.197,E2 16387.197} C_VEL
LIN {X 0,Y 347.81,Z 431.762,A -85,B 0,C 180,E1 16381.976,E2 16381.976} C_VEL
LIN {X 0,Y 347.008,Z 430.351,A -85,B 0,C 180,E1 16379.669,E2 16379.669} C_VEL
LIN {X 0,Y 346.119,Z 429.718,A -85,B 0,C 180,E1 16374.197,E2 16374.197} C_VEL
LIN {X 0,Y 347.073,Z 430.612,A -85,B 0,C 180,E1 16369.543,E2 16369.543} C_VEL
LIN {X 0,Y 350.468,Z 436.396,A -85,B 0,C 180,E1 16362.74,E2 16362.74} C_VEL
LIN {X 0,Y 352.342,Z 440.209,A -85,B 0,C 180,E1 16360.09,E2 16360.09} C_VEL
LIN {X 0,Y 353.495,Z 441.637,A -85,B 0,C 180,E1 16358.947,E2 16358.947} C_VEL
LIN {X 0,Y 355.646,Z 445.733,A -85,B 0,C 180,E1 16356.646,E2 16356.646} C_VEL
LIN {X 0,Y 356.503,Z 447.258,A -85,B 0,C 180,E1 16355.828,E2 16355.828} C_VEL
LIN {X 0,Y 359.308,Z 452.327,A -85,B 0,C 180,E1 16353.383,E2 16353.383} C_VEL
LIN {X 0,Y 361.94,Z 457.305,A -85,B 0,C 180,E1 16351.27,E2 16351.27} C_VEL
LIN {X 0,Y 365.988,Z 465.099,A -85,B 0,C 180,E1 16348.363,E2 16348.363} C_VEL
LIN {X 0,Y 368.333,Z 469.499,A -85,B 0,C 180,E1 16346.983,E2 16346.983} C_VEL
LIN {X 0,Y 377.973,Z 483.118,A -85,B 0,C 180,E1 16343.798,E2 16343.798} C_VEL
LIN {X 0,Y 386.308,Z 495.709,A -85,B 0,C 180,E1 16341.36,E2 16341.36} C_VEL
LIN {X 0,Y 394.671,Z 509.31,A -85,B 0,C 180,E1 16339.137,E2 16339.137} C_VEL
LIN {X 0,Y 395.894,Z 521.794,A -85,B 0,C 180,E1 16338.534,E2 16338.534} C_VEL
LIN {X 0,Y 386.055,Z 752.618,A -85,B 0,C 180,E1 16334.302,E2 16334.302} C_VEL
LIN {X 0,Y 384.402,Z 773.14,A -85,B 0,C 180,E1 16333.677,E2 16333.677} C_VEL
LIN {X 0,Y 381.881,Z 793.746,A -85,B 0,C 180,E1 16332.8,E2 16332.8} C_VEL
LIN {X 0,Y 378.711,Z 813.264,A -85,B 0,C 180,E1 16331.707,E2 16331.707} C_VEL
LIN {X 0,Y 374.924,Z 831.795,A -85,B 0,C 180,E1 16330.394,E2 16330.394} C_VEL
LIN {X 0,Y 370.615,Z 849.426,A -85,B 0,C 180,E1 16328.848,E2 16328.848} C_VEL
LIN {X 0,Y 365.706,Z 866.935,A -85,B 0,C 180,E1 16326.977,E2 16326.977} C_VEL
LIN {X 0,Y 360.744,Z 882.845,A -85,B 0,C 180,E1 16324.914,E2 16324.914} C_VEL
LIN {X 0,Y 355.798,Z 897.228,A -85,B 0,C 180,E1 16322.654,E2 16322.654} C_VEL
LIN {X 0,Y 350.835,Z 910.685,A -85,B 0,C 180,E1 16320.106,E2 16320.106} C_VEL
LIN {X 0,Y 345.942,Z 923.435,A -85,B 0,C 180,E1 16317.172,E2 16317.172} C_VEL
LIN {X 0,Y 341.767,Z 934.107,A -85,B 0,C 180,E1 16314.179,E2 16314.179} C_VEL
LIN {X 0,Y 337.971,Z 943.823,A -85,B 0,C 180,E1 16310.793,E2 16310.793} C_VEL
LIN {X 0,Y 335.021,Z 951.567,A -85,B 0,C 180,E1 16307.365,E2 16307.365} C_VEL
LIN {X 0,Y 332.766,Z 957.92,A -85,B 0,C 180,E1 16303.732,E2 16303.732} C_VEL
LIN {X 0,Y 331.249,Z 962.794,A -85,B 0,C 180,E1 16299.907,E2 16299.907} C_VEL
LIN {X 0,Y 330.41,Z 965.918,A -85,B 0,C 180,E1 16296.254,E2 16296.254} C_VEL
LIN {X 0,Y 330.01,Z 967.601,A -85,B 0,C 180,E1 16292.431,E2 16292.431} C_VEL
LIN {X 0,Y 329.947,Z 967.813,A -85,B 0,C 180,E1 16288.785,E2 16288.785} C_VEL
LIN {X 0,Y 330.008,Z 967.593,A -85,B 0,C 180,E1 16287.439,E2 16287.439} C_VEL
LIN {X 0,Y 329.109,Z 967.346,A -85,B 0,C 180,E1 16286.1,E2 16286.1} C_VEL
LIN {X 0,Y 323.491,Z 966.44,A -85,B 0,C 180,E1 16282.497,E2 16282.497} C_VEL
LIN {X 0,Y 323.031,Z 965.685,A -85,B 0,C 180,E1 16281.321,E2 16281.321} C_VEL
LIN {X 0,Y 324.274,Z 961.65,A -85,B 0,C 180,E1 16277.535,E2 16277.535} C_VEL
LIN {X 0,Y 326.297,Z 956.068,A -85,B 0,C 180,E1 16273.808,E2 16273.808} C_VEL
LIN {X 0,Y 329.141,Z 948.742,A -85,B 0,C 180,E1 16270.109,E2 16270.109} C_VEL
LIN {X 0,Y 332.785,Z 939.933,A -85,B 0,C 180,E1 16266.634,E2 16266.634} C_VEL
LIN {X 0,Y 337.038,Z 929.614,A -85,B 0,C 180,E1 16263.387,E2 16263.387} C_VEL
LIN {X 0,Y 341.852,Z 917.794,A -85,B 0,C 180,E1 16260.376,E2 16260.376} C_VEL
LIN {X 0,Y 347.14,Z 904.288,A -85,B 0,C 180,E1 16257.557,E2 16257.557} C_VEL
LIN {X 0,Y 352.56,Z 889.633,A -85,B 0,C 180,E1 16255.046,E2 16255.046} C_VEL
LIN {X 0,Y 357.785,Z 874.294,A -85,B 0,C 180,E1 16252.869,E2 16252.869} C_VEL
LIN {X 0,Y 362.832,Z 857.648,A -85,B 0,C 180,E1 16250.936,E2 16250.936} C_VEL
LIN {X 0,Y 367.565,Z 839.928,A -85,B 0,C 180,E1 16249.243,E2 16249.243} C_VEL
LIN {X 0,Y 371.687,Z 822.013,A -85,B 0,C 180,E1 16247.842,E2 16247.842} C_VEL
LIN {X 0,Y 375.324,Z 802.726,A -85,B 0,C 180,E1 16246.639,E2 16246.639} C_VEL
LIN {X 0,Y 378.152,Z 783.066,A -85,B 0,C 180,E1 16245.69,E2 16245.69} C_VEL
LIN {X 0,Y 380.31,Z 761.59,A -85,B 0,C 180,E1 16244.924,E2 16244.924} C_VEL
LIN {X 0,Y 381.55,Z 739.943,A -85,B 0,C 180,E1 16244.41,E2 16244.41} C_VEL
LIN {X 0,Y 391.272,Z 522.153,A -85,B 0,C 180,E1 16240.413,E2 16240.413} C_VEL
LIN {X 0,Y 390.265,Z 513.722,A -85,B 0,C 180,E1 16239.949,E2 16239.949} C_VEL
LIN {X 0,Y 381.695,Z 499.78,A -85,B 0,C 180,E1 16237.568,E2 16237.568} C_VEL
LIN {X 0,Y 373.294,Z 487.034,A -85,B 0,C 180,E1 16234.974,E2 16234.974} C_VEL
LIN {X 0,Y 364.747,Z 474.919,A -85,B 0,C 180,E1 16231.989,E2 16231.989} C_VEL
LIN {X 0,Y 359.561,Z 467.636,A -85,B 0,C 180,E1 16229.818,E2 16229.818} C_VEL
LIN {X 0,Y 356.274,Z 461.225,A -85,B 0,C 180,E1 16227.223,E2 16227.223} C_VEL
LIN {X 0,Y 353.963,Z 456.942,A -85,B 0,C 180,E1 16225.249,E2 16225.249} C_VEL
LIN {X 0,Y 351.77,Z 452.709,A -85,B 0,C 180,E1 16223.095,E2 16223.095} C_VEL
LIN {X 0,Y 349.062,Z 447.761,A -85,B 0,C 180,E1 16220.105,E2 16220.105} C_VEL
LIN {X 0,Y 346.892,Z 444.056,A -85,B 0,C 180,E1 16217.271,E2 16217.271} C_VEL
LIN {X 0,Y 346.314,Z 442.759,A -85,B 0,C 180,E1 16216.264,E2 16216.264} C_VEL
LIN {X 0,Y 343.49,Z 437.709,A -85,B 0,C 180,E1 16209.72,E2 16209.72} C_VEL
LIN {X 0,Y 342.797,Z 437.048,A -85,B 0,C 180,E1 16204.685,E2 16204.685} C_VEL
LIN {X 0,Y 343.903,Z 437.907,A -85,B 0,C 180,E1 16199.834,E2 16199.834} C_VEL
LIN {X 0,Y 347.727,Z 443.915,A -85,B 0,C 180,E1 16192.732,E2 16192.732} C_VEL
LIN {X 0,Y 349.788,Z 447.774,A -85,B 0,C 180,E1 16190.125,E2 16190.125} C_VEL
LIN {X 0,Y 351.165,Z 449.503,A -85,B 0,C 180,E1 16188.837,E2 16188.837} C_VEL
LIN {X 0,Y 353.574,Z 453.571,A -85,B 0,C 180,E1 16186.593,E2 16186.593} C_VEL
LIN {X 0,Y 355.019,Z 456.228,A -85,B 0,C 180,E1 16185.318,E2 16185.318} C_VEL
LIN {X 0,Y 357.56,Z 460.247,A -85,B 0,C 180,E1 16183.428,E2 16183.428} C_VEL
LIN {X 0,Y 360.658,Z 465.716,A -85,B 0,C 180,E1 16181.242,E2 16181.242} C_VEL
LIN {X 0,Y 363.683,Z 469.919,A -85,B 0,C 180,E1 16179.859,E2 16179.859} C_VEL
LIN {X 0,Y 370.714,Z 479.079,A -85,B 0,C 180,E1 16177.314,E2 16177.314} C_VEL
LIN {X 0,Y 380.733,Z 493.157,A -85,B 0,C 180,E1 16174.114,E2 16174.114} C_VEL
LIN {X 0,Y 390.838,Z 508.685,A -85,B 0,C 180,E1 16171.253,E2 16171.253} C_VEL
LIN {X 0,Y 396.642,Z 518.48,A -85,B 0,C 180,E1 16169.73,E2 16169.73} C_VEL
LIN {X 0,Y 385.499,Z 709.843,A -85,B 0,C 180,E1 16165.756,E2 16165.756} C_VEL
LIN {X 0,Y 380.249,Z 798.93,A -85,B 0,C 180,E1 16163.841,E2 16163.841} C_VEL
LIN {X 0,Y 377.556,Z 822.374,A -85,B 0,C 180,E1 16163.14,E2 16163.14} C_VEL
LIN {X 0,Y 373.73,Z 846.598,A -85,B 0,C 180,E1 16162.177,E2 16162.177} C_VEL
LIN {X 0,Y 369.665,Z 868.303,A -85,B 0,C 180,E1 16161.044,E2 16161.044} C_VEL
LIN {X 0,Y 364.926,Z 889.92,A -85,B 0,C 180,E1 16159.614,E2 16159.614} C_VEL
LIN {X 0,Y 359.565,Z 912.144,A -85,B 0,C 180,E1 16157.811,E2 16157.811} C_VEL
LIN {X 0,Y 354.21,Z 932.601,A -85,B 0,C 180,E1 16155.807,E2 16155.807} C_VEL
LIN {X 0,Y 348.747,Z 952.305,A -85,B 0,C 180,E1 16153.479,E2 16153.479} C_VEL
LIN {X 0,Y 343.208,Z 971.911,A -85,B 0,C 180,E1 16150.736,E2 16150.736} C_VEL
LIN {X 0,Y 338.304,Z 989.171,A -85,B 0,C 180,E1 16147.898,E2 16147.898} C_VEL
LIN {X 0,Y 333.734,Z 1005.644,A -85,B 0,C 180,E1 16144.697,E2 16144.697} C_VEL
LIN {X 0,Y 329.755,Z 1020.925,A -85,B 0,C 180,E1 16141.232,E2 16141.232} C_VEL
LIN {X 0,Y 326.708,Z 1033.759,A -85,B 0,C 180,E1 16137.817,E2 16137.817} C_VEL
LIN {X 0,Y 324.208,Z 1045.853,A -85,B 0,C 180,E1 16134.022,E2 16134.022} C_VEL
LIN {X 0,Y 322.616,Z 1055.368,A -85,B 0,C 180,E1 16130.5,E2 16130.5} C_VEL
LIN {X 0,Y 321.556,Z 1063.938,A -85,B 0,C 180,E1 16126.623,E2 16126.623} C_VEL
LIN {X 0,Y 321.051,Z 1070.481,A -85,B 0,C 180,E1 16122.958,E2 16122.958} C_VEL
LIN {X 0,Y 320.88,Z 1075.311,A -85,B 0,C 180,E1 16119.325,E2 16119.325} C_VEL
LIN {X 0,Y 320.949,Z 1078.351,A -85,B 0,C 180,E1 16116.08,E2 16116.08} C_VEL
LIN {X 0,Y 320.99,Z 1080.303,A -85,B 0,C 180,E1 16112.499,E2 16112.499} C_VEL
LIN {X 0,Y 321.008,Z 1080.571,A -85,B 0,C 180,E1 16109.108,E2 16109.108} C_VEL
LIN {X 0,Y 320.988,Z 1079.665,A -85,B 0,C 180,E1 16106.07,E2 16106.07} C_VEL
LIN {X 0,Y 320.891,Z 1077.36,A -85,B 0,C 180,E1 16102.66,E2 16102.66} C_VEL
LIN {X 0,Y 320.93,Z 1073.067,A -85,B 0,C 180,E1 16098.863,E2 16098.863} C_VEL
LIN {X 0,Y 321.203,Z 1067.877,A -85,B 0,C 180,E1 16095.486,E2 16095.486} C_VEL
LIN {X 0,Y 322,Z 1060.08,A -85,B 0,C 180,E1 16091.535,E2 16091.535} C_VEL
LIN {X 0,Y 323.316,Z 1051.076,A -85,B 0,C 180,E1 16087.834,E2 16087.834} C_VEL
LIN {X 0,Y 325.34,Z 1040.194,A -85,B 0,C 180,E1 16084.125,E2 16084.125} C_VEL
LIN {X 0,Y 328.188,Z 1027.447,A -85,B 0,C 180,E1 16080.426,E2 16080.426} C_VEL
LIN {X 0,Y 331.79,Z 1012.981,A -85,B 0,C 180,E1 16076.903,E2 16076.903} C_VEL
LIN {X 0,Y 336.195,Z 996.632,A -85,B 0,C 180,E1 16073.501,E2 16073.501} C_VEL
LIN {X 0,Y 341.058,Z 979.449,A -85,B 0,C 180,E1 16070.445,E2 16070.445} C_VEL
LIN {X 0,Y 346.341,Z 960.756,A -85,B 0,C 180,E1 16067.65,E2 16067.65} C_VEL
LIN {X 0,Y 351.894,Z 940.901,A -85,B 0,C 180,E1 16065.139,E2 16065.139} C_VEL
LIN {X 0,Y 357.158,Z 921.454,A -85,B 0,C 180,E1 16063.057,E2 16063.057} C_VEL
LIN {X 0,Y 362.286,Z 900.845,A -85,B 0,C 180,E1 16061.23,E2 16061.23} C_VEL
LIN {X 0,Y 367.513,Z 878.201,A -85,B 0,C 180,E1 16059.584,E2 16059.584} C_VEL
LIN {X 0,Y 372.012,Z 856.163,A -85,B 0,C 180,E1 16058.296,E2 16058.296} C_VEL
LIN {X 0,Y 375.755,Z 834.266,A -85,B 0,C 180,E1 16057.307,E2 16057.307} C_VEL
LIN {X 0,Y 378.997,Z 810.678,A -85,B 0,C 180,E1 16056.495,E2 16056.495} C_VEL
LIN {X 0,Y 381.018,Z 787.481,A -85,B 0,C 180,E1 16055.898,E2 16055.898} C_VEL
LIN {X 0,Y 392.753,Z 583.905,A -85,B 0,C 180,E1 16051.617,E2 16051.617} C_VEL
LIN {X 0,Y 396.481,Z 518.125,A -85,B 0,C 180,E1 16050.247,E2 16050.247} C_VEL
LIN {X 0,Y 387.419,Z 503.371,A -85,B 0,C 180,E1 16047.847,E2 16047.847} C_VEL
LIN {X 0,Y 378.596,Z 490.306,A -85,B 0,C 180,E1 16045.288,E2 16045.288} C_VEL
LIN {X 0,Y 369.978,Z 478.167,A -85,B 0,C 180,E1 16042.482,E2 16042.482} C_VEL
LIN {X 0,Y 362.522,Z 468.436,A -85,B 0,C 180,E1 16039.746,E2 16039.746} C_VEL
LIN {X 0,Y 360.139,Z 464.684,A -85,B 0,C 180,E1 16038.451,E2 16038.451} C_VEL
LIN {X 0,Y 356.605,Z 458.681,A -85,B 0,C 180,E1 16035.948,E2 16035.948} C_VEL
LIN {X 0,Y 353.665,Z 453.683,A -85,B 0,C 180,E1 16033.571,E2 16033.571} C_VEL
LIN {X 0,Y 351.181,Z 449.661,A -85,B 0,C 180,E1 16031.329,E2 16031.329} C_VEL
LIN {X 0,Y 350.363,Z 448.41,A -85,B 0,C 180,E1 16030.523,E2 16030.523} C_VEL
LIN {X 0,Y 347.873,Z 444.555,A -85,B 0,C 180,E1 16027.763,E2 16027.763} C_VEL
LIN {X 0,Y 347.343,Z 443.349,A -85,B 0,C 180,E1 16026.944,E2 16026.944} C_VEL
LIN {X 0,Y 344.187,Z 438.534,A -85,B 0,C 180,E1 16021.498,E2 16021.498} C_VEL
LIN {X 0,Y 343.336,Z 437.44,A -85,B 0,C 180,E1 16019.165,E2 16019.165} C_VEL
LIN {X 0,Y 342.618,Z 436.903,A -85,B 0,C 180,E1 16013.801,E2 16013.801} C_VEL
LIN {X 0,Y 343.551,Z 437.872,A -85,B 0,C 180,E1 16009.434,E2 16009.434} C_VEL
LIN {X 0,Y 346.681,Z 443.416,A -85,B 0,C 180,E1 16002.891,E2 16002.891} C_VEL
LIN {X 0,Y 348.513,Z 447.194,A -85,B 0,C 180,E1 16000.212,E2 16000.212} C_VEL
LIN {X 0,Y 349.589,Z 448.695,A -85,B 0,C 180,E1 15999.052,E2 15999.052} C_VEL
LIN {X 0,Y 351.951,Z 452.932,A -85,B 0,C 180,E1 15996.563,E2 15996.563} C_VEL
LIN {X 0,Y 355.162,Z 459.159,A -85,B 0,C 180,E1 15993.54,E2 15993.54} C_VEL
LIN {X 0,Y 357.697,Z 464.042,A -85,B 0,C 180,E1 15991.445,E2 15991.445} C_VEL
LIN {X 0,Y 360.431,Z 469.205,A -85,B 0,C 180,E1 15989.538,E2 15989.538} C_VEL
LIN {X 0,Y 366.515,Z 477.503,A -85,B 0,C 180,E1 15987.213,E2 15987.213} C_VEL
LIN {X 0,Y 375.053,Z 489.708,A -85,B 0,C 180,E1 15984.326,E2 15984.326} C_VEL
LIN {X 0,Y 383.138,Z 502.143,A -85,B 0,C 180,E1 15981.889,E2 15981.889} C_VEL
LIN {X 0,Y 390.339,Z 514.084,A -85,B 0,C 180,E1 15979.904,E2 15979.904} C_VEL
LIN {X 0,Y 391.176,Z 523.307,A -85,B 0,C 180,E1 15979.459,E2 15979.459} C_VEL
LIN {X 0,Y 380.845,Z 753.382,A -85,B 0,C 180,E1 15975.202,E2 15975.202} C_VEL
LIN {X 0,Y 379.112,Z 773.976,A -85,B 0,C 180,E1 15974.569,E2 15974.569} C_VEL
LIN {X 0,Y 376.458,Z 794.813,A -85,B 0,C 180,E1 15973.674,E2 15973.674} C_VEL
LIN {X 0,Y 373.17,Z 814.28,A -85,B 0,C 180,E1 15972.574,E2 15972.574} C_VEL
LIN {X 0,Y 369.246,Z 832.801,A -85,B 0,C 180,E1 15971.251,E2 15971.251} C_VEL
LIN {X 0,Y 364.777,Z 850.433,A -85,B 0,C 180,E1 15969.692,E2 15969.692} C_VEL
LIN {X 0,Y 359.685,Z 867.958,A -85,B 0,C 180,E1 15967.803,E2 15967.803} C_VEL
LIN {X 0,Y 354.522,Z 883.891,A -85,B 0,C 180,E1 15965.719,E2 15965.719} C_VEL
LIN {X 0,Y 349.206,Z 898.765,A -85,B 0,C 180,E1 15963.35,E2 15963.35} C_VEL
LIN {X 0,Y 344.038,Z 912.17,A -85,B 0,C 180,E1 15960.764,E2 15960.764} C_VEL
LIN {X 0,Y 338.821,Z 925.153,A -85,B 0,C 180,E1 15957.711,E2 15957.711} C_VEL
LIN {X 0,Y 334.337,Z 936.044,A -85,B 0,C 180,E1 15954.563,E2 15954.563} C_VEL
LIN {X 0,Y 330.401,Z 945.667,A -85,B 0,C 180,E1 15951.108,E2 15951.108} C_VEL
LIN {X 0,Y 327.21,Z 953.676,A -85,B 0,C 180,E1 15947.425,E2 15947.425} C_VEL
LIN {X 0,Y 324.893,Z 959.83,A -85,B 0,C 180,E1 15943.708,E2 15943.708} C_VEL
LIN {X 0,Y 323.347,Z 964.52,A -85,B 0,C 180,E1 15939.792,E2 15939.792} C_VEL
LIN {X 0,Y 322.471,Z 967.568,A -85,B 0,C 180,E1 15935.873,E2 15935.873} C_VEL
LIN {X 0,Y 322.115,Z 969.076,A -85,B 0,C 180,E1 15932.135,E2 15932.135} C_VEL
LIN {X 0,Y 322.07,Z 969.143,A -85,B 0,C 180,E1 15928.399,E2 15928.399} C_VEL
LIN {X 0,Y 322.409,Z 967.813,A -85,B 0,C 180,E1 15924.483,E2 15924.483} C_VEL
LIN {X 0,Y 323.031,Z 965.685,A -85,B 0,C 180,E1 15921.321,E2 15921.321} C_VEL
LIN {X 0,Y 322.438,Z 964.711,A -85,B 0,C 180,E1 15919.958,E2 15919.958} C_VEL
LIN {X 0,Y 317.738,Z 961.669,A -85,B 0,C 180,E1 15916.284,E2 15916.284} C_VEL
LIN {X 0,Y 317.624,Z 960.154,A -85,B 0,C 180,E1 15915.11,E2 15915.11} C_VEL
LIN {X 0,Y 320.281,Z 953.5,A -85,B 0,C 180,E1 15911.243,E2 15911.243} C_VEL
LIN {X 0,Y 323.691,Z 945.526,A -85,B 0,C 180,E1 15907.67,E2 15907.67} C_VEL
LIN {X 0,Y 328.002,Z 935.638,A -85,B 0,C 180,E1 15904.156,E2 15904.156} C_VEL
LIN {X 0,Y 332.99,Z 924.123,A -85,B 0,C 180,E1 15900.893,E2 15900.893} C_VEL
LIN {X 0,Y 338.113,Z 911.74,A -85,B 0,C 180,E1 15898.039,E2 15898.039} C_VEL
LIN {X 0,Y 343.587,Z 897.974,A -85,B 0,C 180,E1 15895.426,E2 15895.426} C_VEL
LIN {X 0,Y 348.99,Z 883.329,A -85,B 0,C 180,E1 15893.114,E2 15893.114} C_VEL
LIN {X 0,Y 354.425,Z 867.121,A -85,B 0,C 180,E1 15891.016,E2 15891.016} C_VEL
LIN {X 0,Y 359.294,Z 850.709,A -85,B 0,C 180,E1 15889.263,E2 15889.263} C_VEL
LIN {X 0,Y 363.932,Z 832.88,A -85,B 0,C 180,E1 15887.692,E2 15887.692} C_VEL
LIN {X 0,Y 368.012,Z 814.24,A -85,B 0,C 180,E1 15886.362,E2 15886.362} C_VEL
LIN {X 0,Y 371.401,Z 794.604,A -85,B 0,C 180,E1 15885.262,E2 15885.262} C_VEL
LIN {X 0,Y 374.109,Z 773.718,A -85,B 0,C 180,E1 15884.376,E2 15884.376} C_VEL
LIN {X 0,Y 375.863,Z 752.979,A -85,B 0,C 180,E1 15883.747,E2 15883.747} C_VEL
LIN {X 0,Y 386.626,Z 523.386,A -85,B 0,C 180,E1 15879.448,E2 15879.448} C_VEL
LIN {X 0,Y 385.988,Z 518.402,A -85,B 0,C 180,E1 15879.155,E2 15879.155} C_VEL
LIN {X 0,Y 377.448,Z 504.479,A -85,B 0,C 180,E1 15876.681,E2 15876.681} C_VEL
LIN {X 0,Y 369.303,Z 491.917,A -85,B 0,C 180,E1 15874.04,E2 15874.04} C_VEL
LIN {X 0,Y 361.7,Z 481.126,A -85,B 0,C 180,E1 15871.266,E2 15871.266} C_VEL
LIN {X 0,Y 355.09,Z 472.165,A -85,B 0,C 180,E1 15868.508,E2 15868.508} C_VEL
LIN {X 0,Y 352.084,Z 467.93,A -85,B 0,C 180,E1 15867.025,E2 15867.025} C_VEL
LIN {X 0,Y 349.83,Z 463.656,A -85,B 0,C 180,E1 15865.025,E2 15865.025} C_VEL
LIN {X 0,Y 347.681,Z 459.451,A -85,B 0,C 180,E1 15862.845,E2 15862.845} C_VEL
LIN {X 0,Y 345.216,Z 454.742,A -85,B 0,C 180,E1 15859.985,E2 15859.985} C_VEL
LIN {X 0,Y 343.097,Z 451.018,A -85,B 0,C 180,E1 15857.085,E2 15857.085} C_VEL
LIN {X 0,Y 342.545,Z 449.784,A -85,B 0,C 180,E1 15856.099,E2 15856.099} C_VEL
LIN {X 0,Y 339.858,Z 444.792,A -85,B 0,C 180,E1 15849.483,E2 15849.483} C_VEL
LIN {X 0,Y 339.307,Z 444.229,A -85,B 0,C 180,E1 15844.225,E2 15844.225} C_VEL
LIN {X 0,Y 340.409,Z 445.186,A -85,B 0,C 180,E1 15839.664,E2 15839.664} C_VEL
LIN {X 0,Y 343.995,Z 450.822,A -85,B 0,C 180,E1 15832.989,E2 15832.989} C_VEL
LIN {X 0,Y 346.012,Z 454.717,A -85,B 0,C 180,E1 15830.352,E2 15830.352} C_VEL
LIN {X 0,Y 347.359,Z 456.447,A -85,B 0,C 180,E1 15829.049,E2 15829.049} C_VEL
LIN {X 0,Y 349.959,Z 460.738,A -85,B 0,C 180,E1 15826.62,E2 15826.62} C_VEL
LIN {X 0,Y 353.739,Z 467.312,A -85,B 0,C 180,E1 15823.582,E2 15823.582} C_VEL
LIN {X 0,Y 360.867,Z 476.322,A -85,B 0,C 180,E1 15820.497,E2 15820.497} C_VEL
LIN {X 0,Y 368.727,Z 486.899,A -85,B 0,C 180,E1 15817.564,E2 15817.564} C_VEL
LIN {X 0,Y 378.078,Z 500.336,A -85,B 0,C 180,E1 15814.507,E2 15814.507} C_VEL
LIN {X 0,Y 387.913,Z 515.757,A -85,B 0,C 180,E1 15811.647,E2 15811.647} C_VEL
LIN {X 0,Y 391.753,Z 522.539,A -85,B 0,C 180,E1 15810.597,E2 15810.597} C_VEL
LIN {X 0,Y 380.118,Z 715.327,A -85,B 0,C 180,E1 15806.572,E2 15806.572} C_VEL
LIN {X 0,Y 375.031,Z 798.416,A -85,B 0,C 180,E1 15804.772,E2 15804.772} C_VEL
LIN {X 0,Y 372.237,Z 821.948,A -85,B 0,C 180,E1 15804.063,E2 15804.063} C_VEL
LIN {X 0,Y 368.256,Z 846.213,A -85,B 0,C 180,E1 15803.093,E2 15803.093} C_VEL
LIN {X 0,Y 363.991,Z 868.126,A -85,B 0,C 180,E1 15801.941,E2 15801.941} C_VEL
LIN {X 0,Y 359.012,Z 889.873,A -85,B 0,C 180,E1 15800.485,E2 15800.485} C_VEL
LIN {X 0,Y 353.398,Z 912.111,A -85,B 0,C 180,E1 15798.651,E2 15798.651} C_VEL
LIN {X 0,Y 347.89,Z 932.266,A -85,B 0,C 180,E1 15796.647,E2 15796.647} C_VEL
LIN {X 0,Y 342.151,Z 951.949,A -85,B 0,C 180,E1 15794.279,E2 15794.279} C_VEL
LIN {X 0,Y 336.331,Z 971.51,A -85,B 0,C 180,E1 15791.484,E2 15791.484} C_VEL
LIN {X 0,Y 331.115,Z 988.961,A -85,B 0,C 180,E1 15788.548,E2 15788.548} C_VEL
LIN {X 0,Y 326.445,Z 1004.867,A -85,B 0,C 180,E1 15785.372,E2 15785.372} C_VEL
LIN {X 0,Y 322.06,Z 1020.779,A -85,B 0,C 180,E1 15781.647,E2 15781.647} C_VEL
LIN {X 0,Y 318.825,Z 1033.817,A -85,B 0,C 180,E1 15778.061,E2 15778.061} C_VEL
LIN {X 0,Y 316.306,Z 1045.394,A -85,B 0,C 180,E1 15774.264,E2 15774.264} C_VEL
LIN {X 0,Y 314.597,Z 1055.233,A -85,B 0,C 180,E1 15770.463,E2 15770.463} C_VEL
LIN {X 0,Y 313.625,Z 1062.834,A -85,B 0,C 180,E1 15766.865,E2 15766.865} C_VEL
LIN {X 0,Y 313.113,Z 1069.348,A -85,B 0,C 180,E1 15763.104,E2 15763.104} C_VEL
LIN {X 0,Y 312.958,Z 1074.104,A -85,B 0,C 180,E1 15759.378,E2 15759.378} C_VEL
LIN {X 0,Y 313.038,Z 1076.966,A -85,B 0,C 180,E1 15756.235,E2 15756.235} C_VEL
LIN {X 0,Y 313.099,Z 1078.934,A -85,B 0,C 180,E1 15752.562,E2 15752.562} C_VEL
LIN {X 0,Y 313.126,Z 1079.205,A -85,B 0,C 180,E1 15749.085,E2 15749.085} C_VEL
LIN {X 0,Y 313.096,Z 1078.292,A -85,B 0,C 180,E1 15745.971,E2 15745.971} C_VEL
LIN {X 0,Y 312.989,Z 1075.972,A -85,B 0,C 180,E1 15742.474,E2 15742.474} C_VEL
LIN {X 0,Y 313,Z 1071.836,A -85,B 0,C 180,E1 15738.719,E2 15738.719} C_VEL
LIN {X 0,Y 313.256,Z 1066.896,A -85,B 0,C 180,E1 15735.395,E2 15735.395} C_VEL
LIN {X 0,Y 314.036,Z 1059.429,A -85,B 0,C 180,E1 15731.434,E2 15731.434} C_VEL
LIN {X 0,Y 315.385,Z 1050.518,A -85,B 0,C 180,E1 15727.639,E2 15727.639} C_VEL
LIN {X 0,Y 317.605,Z 1039.234,A -85,B 0,C 180,E1 15723.648,E2 15723.648} C_VEL
LIN {X 0,Y 320.603,Z 1026.541,A -85,B 0,C 180,E1 15719.86,E2 15719.86} C_VEL
LIN {X 0,Y 324.356,Z 1012.31,A -85,B 0,C 180,E1 15716.298,E2 15716.298} C_VEL
LIN {X 0,Y 329.109,Z 995.666,A -85,B 0,C 180,E1 15712.747,E2 15712.747} C_VEL
LIN {X 0,Y 334.225,Z 978.505,A -85,B 0,C 180,E1 15709.633,E2 15709.633} C_VEL
LIN {X 0,Y 339.55,Z 960.63,A -85,B 0,C 180,E1 15706.908,E2 15706.908} C_VEL
LIN {X 0,Y 345.563,Z 940.133,A -85,B 0,C 180,E1 15704.264,E2 15704.264} C_VEL
LIN {X 0,Y 351.246,Z 920.06,A -85,B 0,C 180,E1 15702.096,E2 15702.096} C_VEL
LIN {X 0,Y 356.527,Z 899.734,A -85,B 0,C 180,E1 15700.287,E2 15700.287} C_VEL
LIN {X 0,Y 361.997,Z 876.908,A -85,B 0,C 180,E1 15698.625,E2 15698.625} C_VEL
LIN {X 0,Y 366.479,Z 855.696,A -85,B 0,C 180,E1 15697.381,E2 15697.381} C_VEL
LIN {X 0,Y 370.392,Z 833.686,A -85,B 0,C 180,E1 15696.381,E2 15696.381} C_VEL
LIN {X 0,Y 373.705,Z 810.411,A -85,B 0,C 180,E1 15695.574,E2 15695.574} C_VEL
LIN {X 0,Y 375.804,Z 787.231,A -85,B 0,C 180,E1 15694.973,E2 15694.973} C_VEL
LIN {X 0,Y 387.816,Z 586.239,A -85,B 0,C 180,E1 15690.722,E2 15690.722} C_VEL
LIN {X 0,Y 391.606,Z 522.013,A -85,B 0,C 180,E1 15689.378,E2 15689.378} C_VEL
LIN {X 0,Y 381.784,Z 506.078,A -85,B 0,C 180,E1 15686.646,E2 15686.646} C_VEL
LIN {X 0,Y 373.388,Z 493.575,A -85,B 0,C 180,E1 15684.055,E2 15684.055} C_VEL
LIN {X 0,Y 364.341,Z 480.92,A -85,B 0,C 180,E1 15680.901,E2 15680.901} C_VEL
LIN {X 0,Y 356.078,Z 470.345,A -85,B 0,C 180,E1 15677.569,E2 15677.569} C_VEL
LIN {X 0,Y 353.095,Z 466.059,A -85,B 0,C 180,E1 15676.026,E2 15676.026} C_VEL
LIN {X 0,Y 349.616,Z 460.383,A -85,B 0,C 180,E1 15673.225,E2 15673.225} C_VEL
LIN {X 0,Y 346.753,Z 455.546,A -85,B 0,C 180,E1 15670.466,E2 15670.466} C_VEL
LIN {X 0,Y 344.145,Z 451.468,A -85,B 0,C 180,E1 15667.512,E2 15667.512} C_VEL
LIN {X 0,Y 343.574,Z 450.342,A -85,B 0,C 180,E1 15666.684,E2 15666.684} C_VEL
LIN {X 0,Y 340.259,Z 444.982,A -85,B 0,C 180,E1 15660.336,E2 15660.336} C_VEL
LIN {X 0,Y 339.059,Z 444.076,A -85,B 0,C 180,E1 15655.094,E2 15655.094} C_VEL
LIN {X 0,Y 339.855,Z 444.766,A -85,B 0,C 180,E1 15650.004,E2 15650.004} C_VEL
LIN {X 0,Y 342.9,Z 450.438,A -85,B 0,C 180,E1 15643.046,E2 15643.046} C_VEL
LIN {X 0,Y 344.832,Z 454.351,A -85,B 0,C 180,E1 15640.168,E2 15640.168} C_VEL
LIN {X 0,Y 345.698,Z 455.75,A -85,B 0,C 180,E1 15639.16,E2 15639.16} C_VEL
LIN {X 0,Y 348.291,Z 460.7,A -85,B 0,C 180,E1 15636.302,E2 15636.302} C_VEL
LIN {X 0,Y 350.927,Z 465.771,A -85,B 0,C 180,E1 15633.792,E2 15633.792} C_VEL
LIN {X 0,Y 353.2,Z 469.546,A -85,B 0,C 180,E1 15632.2,E2 15632.2} C_VEL
LIN {X 0,Y 360.545,Z 479.564,A -85,B 0,C 180,E1 15629.04,E2 15629.04} C_VEL
LIN {X 0,Y 367.031,Z 488.666,A -85,B 0,C 180,E1 15626.613,E2 15626.613} C_VEL
LIN {X 0,Y 375.138,Z 500.8,A -85,B 0,C 180,E1 15623.911,E2 15623.911} C_VEL
LIN {X 0,Y 383.994,Z 515.146,A -85,B 0,C 180,E1 15621.275,E2 15621.275} C_VEL
LIN {X 0,Y 386.102,Z 519.045,A -85,B 0,C 180,E1 15620.68,E2 15620.68} C_VEL
LIN {X 0,Y 386.543,Z 525.076,A -85,B 0,C 180,E1 15620.4,E2 15620.4} C_VEL
LIN {X 0,Y 375.735,Z 754.003,A -85,B 0,C 180,E1 15616.129,E2 15616.129} C_VEL
LIN {X 0,Y 373.939,Z 774.592,A -85,B 0,C 180,E1 15615.494,E2 15615.494} C_VEL
LIN {X 0,Y 371.125,Z 795.869,A -85,B 0,C 180,E1 15614.574,E2 15614.574} C_VEL
LIN {X 0,Y 367.717,Z 815.294,A -85,B 0,C 180,E1 15613.467,E2 15613.467} C_VEL
LIN {X 0,Y 363.653,Z 833.806,A -85,B 0,C 180,E1 15612.135,E2 15612.135} C_VEL
LIN {X 0,Y 359.036,Z 851.386,A -85,B 0,C 180,E1 15610.569,E2 15610.569} C_VEL
LIN {X 0,Y 353.741,Z 868.971,A -85,B 0,C 180,E1 15608.658,E2 15608.658} C_VEL
LIN {X 0,Y 348.566,Z 884.406,A -85,B 0,C 180,E1 15606.63,E2 15606.63} C_VEL
LIN {X 0,Y 343.019,Z 899.351,A -85,B 0,C 180,E1 15604.234,E2 15604.234} C_VEL
LIN {X 0,Y 337.6,Z 912.872,A -85,B 0,C 180,E1 15601.616,E2 15601.616} C_VEL
LIN {X 0,Y 332.246,Z 925.687,A -85,B 0,C 180,E1 15598.587,E2 15598.587} C_VEL
LIN {X 0,Y 327.628,Z 936.43,A -85,B 0,C 180,E1 15595.487,E2 15595.487} C_VEL
LIN {X 0,Y 323.357,Z 946.291,A -85,B 0,C 180,E1 15591.929,E2 15591.929} C_VEL
LIN {X 0,Y 320.058,Z 954.008,A -85,B 0,C 180,E1 15588.393,E2 15588.393} C_VEL
LIN {X 0,Y 317.501,Z 960.427,A -85,B 0,C 180,E1 15584.592,E2 15584.592} C_VEL
LIN {X 0,Y 315.8,Z 965.196,A -85,B 0,C 180,E1 15580.766,E2 15580.766} C_VEL
LIN {X 0,Y 314.753,Z 968.553,A -85,B 0,C 180,E1 15576.75,E2 15576.75} C_VEL
LIN {X 0,Y 314.261,Z 970.277,A -85,B 0,C 180,E1 15572.735,E2 15572.735} C_VEL
LIN {X 0,Y 314.182,Z 970.562,A -85,B 0,C 180,E1 15568.906,E2 15568.906} C_VEL
LIN {X 0,Y 314.479,Z 969.467,A -85,B 0,C 180,E1 15564.893,E2 15564.893} C_VEL
LIN {X 0,Y 315.279,Z 966.875,A -85,B 0,C 180,E1 15560.876,E2 15560.876} C_VEL
LIN {X 0,Y 316.715,Z 962.593,A -85,B 0,C 180,E1 15556.862,E2 15556.862} C_VEL
LIN {X 0,Y 317.624,Z 960.154,A -85,B 0,C 180,E1 15555.11,E2 15555.11} C_VEL
LIN {X 0,Y 317.482,Z 958.338,A -85,B 0,C 180,E1 15553.748,E2 15553.748} C_VEL
LIN {X 0,Y 314.166,Z 953.298,A -85,B 0,C 180,E1 15550.05,E2 15550.05} C_VEL
LIN {X 0,Y 314.49,Z 951.056,A -85,B 0,C 180,E1 15548.907,E2 15548.907} C_VEL
LIN {X 0,Y 318.519,Z 942.256,A -85,B 0,C 180,E1 15545.323,E2 15545.323} C_VEL
LIN {X 0,Y 323.249,Z 931.885,A -85,B 0,C 180,E1 15541.955,E2 15541.955} C_VEL
LIN {X 0,Y 328.534,Z 919.993,A -85,B 0,C 180,E1 15538.843,E2 15538.843} C_VEL
LIN {X 0,Y 334.299,Z 906.433,A -85,B 0,C 180,E1 15535.944,E2 15535.944} C_VEL
LIN {X 0,Y 340.235,Z 891.585,A -85,B 0,C 180,E1 15533.349,E2 15533.349} C_VEL
LIN {X 0,Y 345.833,Z 876.321,A -85,B 0,C 180,E1 15531.142,E2 15531.142} C_VEL
LIN {X 0,Y 351.19,Z 859.894,A -85,B 0,C 180,E1 15529.201,E2 15529.201} C_VEL
LIN {X 0,Y 356.357,Z 841.897,A -85,B 0,C 180,E1 15527.453,E2 15527.453} C_VEL
LIN {X 0,Y 360.78,Z 823.994,A -85,B 0,C 180,E1 15526.034,E2 15526.034} C_VEL
LIN {X 0,Y 364.588,Z 805.18,A -85,B 0,C 180,E1 15524.841,E2 15524.841} C_VEL
LIN {X 0,Y 367.686,Z 785.423,A -85,B 0,C 180,E1 15523.866,E2 15523.866} C_VEL
LIN {X 0,Y 370.002,Z 764.751,A -85,B 0,C 180,E1 15523.102,E2 15523.102} C_VEL
LIN {X 0,Y 371.401,Z 743.728,A -85,B 0,C 180,E1 15522.572,E2 15522.572} C_VEL
LIN {X 0,Y 382.138,Z 525.213,A -85,B 0,C 180,E1 15518.492,E2 15518.492} C_VEL
LIN {X 0,Y 381.781,Z 523.112,A -85,B 0,C 180,E1 15518.343,E2 15518.343} C_VEL
LIN {X 0,Y 372.547,Z 507.78,A -85,B 0,C 180,E1 15515.525,E2 15515.525} C_VEL
LIN {X 0,Y 364.098,Z 494.91,A -85,B 0,C 180,E1 15512.611,E2 15512.611} C_VEL
LIN {X 0,Y 357.077,Z 484.9,A -85,B 0,C 180,E1 15509.85,E2 15509.85} C_VEL
LIN {X 0,Y 350.228,Z 475.494,A -85,B 0,C 180,E1 15506.721,E2 15506.721} C_VEL
LIN {X 0,Y 345.709,Z 469.838,A -85,B 0,C 180,E1 15504.34,E2 15504.34} C_VEL
